LIN {X -90.429,Y -7.308,Z -76.160,A -90.000,B 90.000,C 0.000} C_DIS
LIN {X -90.430,Y -7.308,Z -76.160,A -90.000,B 90.000,C 0.000} C_DIS
LIN {X -90.438,Y -7.308,Z -76.159,A -90.000,B 90.000,C 0.000} C_DIS
LIN {X -90.556,Y -7.308,Z -76.141,A -90.000,B 90.000,C 0.000} C_DIS
LIN {X -90.743,Y -7.308,Z -76.119,A -90.000,B 90.000,C 0.000} C_DIS
LIN {X -90.835,Y -7.308,Z -76.112,A -90.000,B 90.000,C 0.000} C_DIS
LIN {X -90.996,Y -7.308,Z -76.109,A -90.000,B 90.000,C 0.000} C_DIS
LIN {X -91.021,Y -7.308,Z -76.109,A -90.000,B 90.000,C 0.000} C_DIS
LIN {X -91.083,Y -7.308,Z -76.111,A -90.000,B 90.000,C 0.000} C_DIS
LIN {X -91.127,Y -7.308,Z -76.111,A -90.000,B 90.000,C 0.000} C_DIS
LIN {X -91.716,Y -7.308,Z -76.119,A -90.000,B 90.000,C 0.000} C_DIS
LIN {X -91.719,Y -7.308,Z -76.119,A -90.000,B 90.000,C 0.000} C_DIS
LIN {X -91.850,Y -7.308,Z -76.127,A -90.000,B 90.000,C 0.000} C_DIS
LIN {X -91.854,Y -7.308,Z -76.127,A -90.000,B 90.000,C 0.000} C_DIS
LIN {X -91.855,Y -7.308,Z -76.127,A -90.000,B 90.000,C 0.000} C_DIS
LIN {X -92.275,Y -7.308,Z -76.134,A -90.000,B 90.000,C 0.000} C_DIS
LIN {X -92.401,Y -7.308,Z -76.144,A -90.000,B 90.000,C 0.000} C_DIS
LIN {X -92.567,Y -7.308,Z -76.154,A -90.000,B 90.000,C 0.000} C_DIS
LIN {X -92.855,Y -7.308,Z -76.172,A -90.000,B 90.000,C 0.000} C_DIS
LIN {X -93.155,Y -7.308,Z -76.171,A -90.000,B 90.000,C 0.000} C_DIS
LIN {X -93.950,Y -7.308,Z -76.211,A -90.000,B 90.000,C 0.000} C_DIS
LIN {X -93.975,Y -7.308,Z -76.209,A -90.000,B 90.000,C 0.000} C_DIS
LIN {X -94.009,Y -7.308,Z -76.208,A -90.000,B 90.000,C 0.000} C_DIS
LIN {X -94.203,Y -7.308,Z -76.206,A -90.000,B 90.000,C 0.000} C_DIS
LIN {X -94.938,Y -7.308,Z -76.181,A -90.000,B 90.000,C 0.000} C_DIS
LIN {X -95.138,Y -7.308,Z -76.181,A -90.000,B 90.000,C 0.000} C_DIS
LIN {X -95.500,Y -7.308,Z -76.164,A -90.000,B 90.000,C 0.000} C_DIS
LIN {X -95.593,Y -7.308,Z -76.159,A -90.000,B 90.000,C 0.000} C_DIS
LIN {X -96.438,Y -7.308,Z -76.050,A -90.000,B 90.000,C 0.000} C_DIS
LIN {X -96.876,Y -7.308,Z -76.007,A -90.000,B 90.000,C 0.000} C_DIS
LIN {X -97.150,Y -7.308,Z -75.964,A -90.000,B 90.000,C 0.000} C_DIS
LIN {X -97.326,Y -7.308,Z -75.936,A -90.000,B 90.000,C 0.000} C_DIS
LIN {X -98.066,Y -7.308,Z -75.745,A -90.000,B 90.000,C 0.000} C_DIS
LIN {X -98.704,Y -7.308,Z -75.598,A -90.000,B 90.000,C 0.000} C_DIS
LIN {X -98.924,Y -7.308,Z -75.538,A -90.000,B 90.000,C 0.000} C_DIS
LIN {X -99.143,Y -7.308,Z -75.478,A -90.000,B 90.000,C 0.000} C_DIS
LIN {X -99.355,Y -7.308,Z -75.394,A -90.000,B 90.000,C 0.000} C_DIS
LIN {X -99.566,Y -7.308,Z -75.311,A -90.000,B 90.000,C 0.000} C_DIS
LIN {X -100.148,Y -7.308,Z -75.070,A -90.000,B 90.000,C 0.000} C_DIS
LIN {X -100.612,Y -7.308,Z -74.890,A -90.000,B 90.000,C 0.000} C_DIS
LIN {X -100.815,Y -7.308,Z -74.810,A -90.000,B 90.000,C 0.000} C_DIS
LIN {X -101.035,Y -7.308,Z -74.723,A -90.000,B 90.000,C 0.000} C_DIS
LIN {X -101.228,Y -7.308,Z -74.620,A -90.000,B 90.000,C 0.000} C_DIS
LIN {X -101.438,Y -7.308,Z -74.510,A -90.000,B 90.000,C 0.000} C_DIS
LIN {X -102.233,Y -7.308,Z -74.035,A -90.000,B 90.000,C 0.000} C_DIS
LIN {X -102.984,Y -7.308,Z -73.608,A -90.000,B 90.000,C 0.000} C_DIS
LIN {X -103.195,Y -7.308,Z -73.465,A -90.000,B 90.000,C 0.000} C_DIS
LIN {X -103.361,Y -7.308,Z -73.353,A -90.000,B 90.000,C 0.000} C_DIS
LIN {X -104.367,Y -7.308,Z -72.602,A -90.000,B 90.000,C 0.000} C_DIS
LIN {X -104.886,Y -7.308,Z -72.231,A -90.000,B 90.000,C 0.000} C_DIS
LIN {X -105.135,Y -7.308,Z -72.019,A -90.000,B 90.000,C 0.000} C_DIS
LIN {X -105.233,Y -7.308,Z -71.935,A -90.000,B 90.000,C 0.000} C_DIS
LIN {X -106.016,Y -7.308,Z -71.241,A -90.000,B 90.000,C 0.000} C_DIS
LIN {X -106.511,Y -7.308,Z -70.803,A -90.000,B 90.000,C 0.000} C_DIS
LIN {X -106.623,Y -7.308,Z -70.708,A -90.000,B 90.000,C 0.000} C_DIS
LIN {X -106.647,Y -7.308,Z -70.687,A -90.000,B 90.000,C 0.000} C_DIS
LIN {X -107.011,Y -7.308,Z -70.310,A -90.000,B 90.000,C 0.000} C_DIS
LIN {X -107.247,Y -7.308,Z -70.060,A -90.000,B 90.000,C 0.000} C_DIS
LIN {X -107.570,Y -7.308,Z -69.717,A -90.000,B 90.000,C 0.000} C_DIS
LIN {X -107.658,Y -7.308,Z -69.623,A -90.000,B 90.000,C 0.000} C_DIS
LIN {X -107.961,Y -7.308,Z -69.302,A -90.000,B 90.000,C 0.000} C_DIS
LIN {X -108.119,Y -7.308,Z -69.134,A -90.000,B 90.000,C 0.000} C_DIS
LIN {X -108.189,Y -7.308,Z -69.054,A -90.000,B 90.000,C 0.000} C_DIS
LIN {X -108.324,Y -7.308,Z -68.876,A -90.000,B 90.000,C 0.000} C_DIS
LIN {X -108.394,Y -7.308,Z -68.788,A -90.000,B 90.000,C 0.000} C_DIS
LIN {X -108.549,Y -7.308,Z -68.594,A -90.000,B 90.000,C 0.000} C_DIS
LIN {X -108.807,Y -7.308,Z -68.269,A -90.000,B 90.000,C 0.000} C_DIS
LIN {X -109.048,Y -7.308,Z -67.965,A -90.000,B 90.000,C 0.000} C_DIS
LIN {X -109.050,Y -7.308,Z -67.962,A -90.000,B 90.000,C 0.000} C_DIS
LIN {X -109.051,Y -7.308,Z -67.961,A -90.000,B 90.000,C 0.000} C_DIS
LIN {X -109.057,Y -7.308,Z -67.953,A -90.000,B 90.000,C 0.000} C_DIS
LIN {X -109.064,Y -7.308,Z -67.944,A -90.000,B 90.000,C 0.000} C_DIS
LIN {X -109.315,Y -7.308,Z -67.619,A -90.000,B 90.000,C 0.000} C_DIS
LIN {X -109.317,Y -7.308,Z -67.616,A -90.000,B 90.000,C 0.000} C_DIS
LIN {X -109.330,Y -7.308,Z -67.598,A -90.000,B 90.000,C 0.000} C_DIS
LIN {X -109.445,Y -7.308,Z -67.437,A -90.000,B 90.000,C 0.000} C_DIS
LIN {X -109.557,Y -7.308,Z -67.257,A -90.000,B 90.000,C 0.000} C_DIS
LIN {X -109.624,Y -7.308,Z -67.149,A -90.000,B 90.000,C 0.000} C_DIS
LIN {X -109.859,Y -7.308,Z -66.772,A -90.000,B 90.000,C 0.000} C_DIS
LIN {X -110.128,Y -7.308,Z -66.355,A -90.000,B 90.000,C 0.000} C_DIS
LIN {X -110.187,Y -7.308,Z -66.262,A -90.000,B 90.000,C 0.000} C_DIS
LIN {X -110.241,Y -7.308,Z -66.176,A -90.000,B 90.000,C 0.000} C_DIS
LIN {X -110.406,Y -7.308,Z -65.897,A -90.000,B 90.000,C 0.000} C_DIS
LIN {X -110.474,Y -7.308,Z -65.784,A -90.000,B 90.000,C 0.000} C_DIS
LIN {X -111.122,Y -7.308,Z -64.499,A -90.000,B 90.000,C 0.000} C_DIS
LIN {X -111.141,Y -7.308,Z -64.462,A -90.000,B 90.000,C 0.000} C_DIS
LIN {X -111.142,Y -7.308,Z -64.459,A -90.000,B 90.000,C 0.000} C_DIS
LIN {X -111.143,Y -7.308,Z -64.457,A -90.000,B 90.000,C 0.000} C_DIS
LIN {X -111.144,Y -7.308,Z -64.456,A -90.000,B 90.000,C 0.000} C_DIS
LIN {X -111.144,Y -7.308,Z -64.455,A -90.000,B 90.000,C 0.000} C_DIS
LIN {X -111.330,Y -7.308,Z -64.046,A -90.000,B 90.000,C 0.000} C_DIS
LIN {X -111.330,Y -7.308,Z -64.044,A -90.000,B 90.000,C 0.000} C_DIS
LIN {X -111.331,Y -7.308,Z -64.041,A -90.000,B 90.000,C 0.000} C_DIS
LIN {X -111.339,Y -7.308,Z -64.023,A -90.000,B 90.000,C 0.000} C_DIS
LIN {X -111.858,Y -7.308,Z -62.803,A -90.000,B 90.000,C 0.000} C_DIS
LIN {X -111.946,Y -7.308,Z -62.595,A -90.000,B 90.000,C 0.000} C_DIS
LIN {X -111.980,Y -7.308,Z -62.501,A -90.000,B 90.000,C 0.000} C_DIS
LIN {X -112.247,Y -7.308,Z -61.757,A -90.000,B 90.000,C 0.000} C_DIS
LIN {X -112.297,Y -7.308,Z -61.622,A -90.000,B 90.000,C 0.000} C_DIS
LIN {X -112.357,Y -7.308,Z -61.457,A -90.000,B 90.000,C 0.000} C_DIS
LIN {X -112.381,Y -7.308,Z -61.394,A -90.000,B 90.000,C 0.000} C_DIS
LIN {X -112.489,Y -7.308,Z -61.121,A -90.000,B 90.000,C 0.000} C_DIS
LIN {X -112.498,Y -7.308,Z -61.099,A -90.000,B 90.000,C 0.000} C_DIS
LIN {X -112.511,Y -7.308,Z -61.065,A -90.000,B 90.000,C 0.000} C_DIS
LIN {X -112.548,Y -7.308,Z -60.970,A -90.000,B 90.000,C 0.000} C_DIS
LIN {X -112.569,Y -7.308,Z -60.913,A -90.000,B 90.000,C 0.000} C_DIS
LIN {X -112.574,Y -7.308,Z -60.900,A -90.000,B 90.000,C 0.000} C_DIS
LIN {X -112.579,Y -7.308,Z -60.889,A -90.000,B 90.000,C 0.000} C_DIS
LIN {X -112.589,Y -7.308,Z -60.860,A -90.000,B 90.000,C 0.000} C_DIS
LIN {X -112.641,Y -7.308,Z -60.721,A -90.000,B 90.000,C 0.000} C_DIS
LIN {X -112.737,Y -7.308,Z -60.464,A -90.000,B 90.000,C 0.000} C_DIS
LIN {X -112.752,Y -7.308,Z -60.423,A -90.000,B 90.000,C 0.000} C_DIS
LIN {X -112.766,Y -7.308,Z -60.386,A -90.000,B 90.000,C 0.000} C_DIS
LIN {X -112.917,Y -7.308,Z -59.968,A -90.000,B 90.000,C 0.000} C_DIS
LIN {X -112.929,Y -7.308,Z -59.935,A -90.000,B 90.000,C 0.000} C_DIS
LIN {X -112.957,Y -7.308,Z -59.850,A -90.000,B 90.000,C 0.000} C_DIS
LIN {X -113.226,Y -7.308,Z -59.066,A -90.000,B 90.000,C 0.000} C_DIS
LIN {X -113.275,Y -7.308,Z -58.928,A -90.000,B 90.000,C 0.000} C_DIS
LIN {X -113.292,Y -7.308,Z -58.880,A -90.000,B 90.000,C 0.000} C_DIS
LIN {X -113.430,Y -7.308,Z -58.480,A -90.000,B 90.000,C 0.000} C_DIS
LIN {X -113.480,Y -7.308,Z -58.334,A -90.000,B 90.000,C 0.000} C_DIS
LIN {X -113.651,Y -7.308,Z -57.841,A -90.000,B 90.000,C 0.000} C_DIS
LIN {X -113.725,Y -7.308,Z -57.605,A -90.000,B 90.000,C 0.000} C_DIS
LIN {X -113.775,Y -7.308,Z -57.446,A -90.000,B 90.000,C 0.000} C_DIS
LIN {X -113.840,Y -7.308,Z -57.265,A -90.000,B 90.000,C 0.000} C_DIS
LIN {X -113.863,Y -7.308,Z -57.201,A -90.000,B 90.000,C 0.000} C_DIS
LIN {X -113.998,Y -7.308,Z -56.823,A -90.000,B 90.000,C 0.000} C_DIS
LIN {X -114.035,Y -7.308,Z -56.712,A -90.000,B 90.000,C 0.000} C_DIS
LIN {X -114.077,Y -7.308,Z -56.590,A -90.000,B 90.000,C 0.000} C_DIS
LIN {X -114.087,Y -7.308,Z -56.561,A -90.000,B 90.000,C 0.000} C_DIS
LIN {X -114.176,Y -7.308,Z -56.299,A -90.000,B 90.000,C 0.000} C_DIS
LIN {X -114.177,Y -7.308,Z -56.295,A -90.000,B 90.000,C 0.000} C_DIS
LIN {X -114.260,Y -7.308,Z -56.079,A -90.000,B 90.000,C 0.000} C_DIS
LIN {X -114.595,Y -7.308,Z -55.238,A -90.000,B 90.000,C 0.000} C_DIS
LIN {X -114.855,Y -7.308,Z -54.587,A -90.000,B 90.000,C 0.000} C_DIS
LIN {X -115.040,Y -7.308,Z -54.138,A -90.000,B 90.000,C 0.000} C_DIS
LIN {X -115.335,Y -7.308,Z -53.342,A -90.000,B 90.000,C 0.000} C_DIS
LIN {X -115.406,Y -7.308,Z -53.154,A -90.000,B 90.000,C 0.000} C_DIS
LIN {X -115.537,Y -7.308,Z -52.781,A -90.000,B 90.000,C 0.000} C_DIS
LIN {X -115.545,Y -7.308,Z -52.758,A -90.000,B 90.000,C 0.000} C_DIS
LIN {X -115.549,Y -7.308,Z -52.745,A -90.000,B 90.000,C 0.000} C_DIS
LIN {X -115.560,Y -7.308,Z -52.713,A -90.000,B 90.000,C 0.000} C_DIS
LIN {X -115.573,Y -7.308,Z -52.666,A -90.000,B 90.000,C 0.000} C_DIS
LIN {X -115.577,Y -7.308,Z -52.655,A -90.000,B 90.000,C 0.000} C_DIS
LIN {X -115.783,Y -7.308,Z -51.915,A -90.000,B 90.000,C 0.000} C_DIS
LIN {X -115.800,Y -7.308,Z -51.855,A -90.000,B 90.000,C 0.000} C_DIS
LIN {X -115.805,Y -7.308,Z -51.837,A -90.000,B 90.000,C 0.000} C_DIS
LIN {X -115.851,Y -7.308,Z -51.672,A -90.000,B 90.000,C 0.000} C_DIS
LIN {X -115.877,Y -7.308,Z -51.578,A -90.000,B 90.000,C 0.000} C_DIS
LIN {X -115.919,Y -7.308,Z -51.379,A -90.000,B 90.000,C 0.000} C_DIS
LIN {X -115.971,Y -7.308,Z -51.132,A -90.000,B 90.000,C 0.000} C_DIS
LIN {X -115.990,Y -7.308,Z -50.930,A -90.000,B 90.000,C 0.000} C_DIS
LIN {X -115.995,Y -7.308,Z -50.884,A -90.000,B 90.000,C 0.000} C_DIS
LIN {X -116.015,Y -7.308,Z -50.679,A -90.000,B 90.000,C 0.000} C_DIS
LIN {X -116.038,Y -7.308,Z -50.413,A -90.000,B 90.000,C 0.000} C_DIS
LIN {X -116.044,Y -7.308,Z -50.351,A -90.000,B 90.000,C 0.000} C_DIS
LIN {X -116.053,Y -7.308,Z -50.262,A -90.000,B 90.000,C 0.000} C_DIS
LIN {X -116.072,Y -7.308,Z -50.070,A -90.000,B 90.000,C 0.000} C_DIS
LIN {X -116.088,Y -7.308,Z -49.898,A -90.000,B 90.000,C 0.000} C_DIS
LIN {X -116.085,Y -7.308,Z -49.616,A -90.000,B 90.000,C 0.000} C_DIS
LIN {X -116.082,Y -7.308,Z -49.442,A -90.000,B 90.000,C 0.000} C_DIS
LIN {X -116.079,Y -7.308,Z -49.392,A -90.000,B 90.000,C 0.000} C_DIS
LIN {X -116.077,Y -7.308,Z -49.365,A -90.000,B 90.000,C 0.000} C_DIS
LIN {X -116.068,Y -7.308,Z -49.205,A -90.000,B 90.000,C 0.000} C_DIS
LIN {X -116.055,Y -7.308,Z -48.764,A -90.000,B 90.000,C 0.000} C_DIS
LIN {X -116.049,Y -7.308,Z -48.715,A -90.000,B 90.000,C 0.000} C_DIS
LIN {X -116.049,Y -7.308,Z -48.713,A -90.000,B 90.000,C 0.000} C_DIS
LIN {X -116.045,Y -7.308,Z -48.687,A -90.000,B 90.000,C 0.000} C_DIS
LIN {X -116.046,Y -7.308,Z -48.684,A -90.000,B 90.000,C 0.000} C_DIS
LIN {X -116.102,Y -7.308,Z -48.546,A -90.000,B 90.000,C 0.000} C_DIS
LIN {X -116.109,Y -7.308,Z -48.529,A -90.000,B 90.000,C 0.000} C_DIS
LIN {X -116.231,Y -7.308,Z -48.216,A -90.000,B 90.000,C 0.000} C_DIS
LIN {X -116.273,Y -7.308,Z -48.106,A -90.000,B 90.000,C 0.000} C_DIS
LIN {X -116.402,Y -7.308,Z -47.760,A -90.000,B 90.000,C 0.000} C_DIS
LIN {X -116.428,Y -7.308,Z -47.687,A -90.000,B 90.000,C 0.000} C_DIS
LIN {X -116.462,Y -7.308,Z -47.594,A -90.000,B 90.000,C 0.000} C_DIS
LIN {X -116.577,Y -7.308,Z -47.256,A -90.000,B 90.000,C 0.000} C_DIS
LIN {X -116.682,Y -7.308,Z -46.928,A -90.000,B 90.000,C 0.000} C_DIS
LIN {X -116.712,Y -7.308,Z -46.836,A -90.000,B 90.000,C 0.000} C_DIS
LIN {X -116.738,Y -7.308,Z -46.742,A -90.000,B 90.000,C 0.000} C_DIS
LIN {X -116.816,Y -7.308,Z -46.454,A -90.000,B 90.000,C 0.000} C_DIS
LIN {X -116.874,Y -7.308,Z -46.240,A -90.000,B 90.000,C 0.000} C_DIS
LIN {X -116.912,Y -7.308,Z -46.079,A -90.000,B 90.000,C 0.000} C_DIS
LIN {X -116.977,Y -7.308,Z -45.819,A -90.000,B 90.000,C 0.000} C_DIS
LIN {X -117.000,Y -7.308,Z -45.688,A -90.000,B 90.000,C 0.000} C_DIS
LIN {X -117.032,Y -7.308,Z -45.502,A -90.000,B 90.000,C 0.000} C_DIS
LIN {X -117.066,Y -7.308,Z -45.295,A -90.000,B 90.000,C 0.000} C_DIS
LIN {X -117.091,Y -7.308,Z -45.116,A -90.000,B 90.000,C 0.000} C_DIS
LIN {X -117.122,Y -7.308,Z -44.884,A -90.000,B 90.000,C 0.000} C_DIS
LIN {X -117.154,Y -7.308,Z -44.619,A -90.000,B 90.000,C 0.000} C_DIS
LIN {X -117.172,Y -7.308,Z -44.476,A -90.000,B 90.000,C 0.000} C_DIS
LIN {X -117.184,Y -7.308,Z -44.378,A -90.000,B 90.000,C 0.000} C_DIS
LIN {X -117.189,Y -7.308,Z -44.049,A -90.000,B 90.000,C 0.000} C_DIS
LIN {X -117.191,Y -7.308,Z -43.922,A -90.000,B 90.000,C 0.000} C_DIS
LIN {X -117.191,Y -7.308,Z -43.911,A -90.000,B 90.000,C 0.000} C_DIS
LIN {X -117.188,Y -7.308,Z -43.790,A -90.000,B 90.000,C 0.000} C_DIS
LIN {X -117.187,Y -7.308,Z -43.750,A -90.000,B 90.000,C 0.000} C_DIS
LIN {X -117.190,Y -7.308,Z -43.518,A -90.000,B 90.000,C 0.000} C_DIS
LIN {X -117.191,Y -7.308,Z -43.491,A -90.000,B 90.000,C 0.000} C_DIS
LIN {X -117.191,Y -7.308,Z -43.489,A -90.000,B 90.000,C 0.000} C_DIS
LIN {X -117.190,Y -7.308,Z -43.459,A -90.000,B 90.000,C 0.000} C_DIS
LIN {X -117.185,Y -7.308,Z -43.036,A -90.000,B 90.000,C 0.000} C_DIS
LIN {X -117.181,Y -7.308,Z -43.004,A -90.000,B 90.000,C 0.000} C_DIS
LIN {X -117.153,Y -7.308,Z -42.780,A -90.000,B 90.000,C 0.000} C_DIS
LIN {X -117.137,Y -7.308,Z -42.642,A -90.000,B 90.000,C 0.000} C_DIS
LIN {X -117.132,Y -7.308,Z -42.602,A -90.000,B 90.000,C 0.000} C_DIS
LIN {X -117.129,Y -7.308,Z -42.575,A -90.000,B 90.000,C 0.000} C_DIS
LIN {X -117.082,Y -7.308,Z -42.199,A -90.000,B 90.000,C 0.000} C_DIS
LIN {X -117.072,Y -7.308,Z -42.126,A -90.000,B 90.000,C 0.000} C_DIS
LIN {X -117.040,Y -7.308,Z -41.945,A -90.000,B 90.000,C 0.000} C_DIS
LIN {X -117.020,Y -7.308,Z -41.836,A -90.000,B 90.000,C 0.000} C_DIS
LIN {X -116.975,Y -7.308,Z -41.649,A -90.000,B 90.000,C 0.000} C_DIS
LIN {X -116.937,Y -7.308,Z -41.456,A -90.000,B 90.000,C 0.000} C_DIS
LIN {X -116.879,Y -7.308,Z -41.233,A -90.000,B 90.000,C 0.000} C_DIS
LIN {X -116.827,Y -7.308,Z -41.029,A -90.000,B 90.000,C 0.000} C_DIS
LIN {X -116.765,Y -7.308,Z -40.854,A -90.000,B 90.000,C 0.000} C_DIS
LIN {X -116.712,Y -7.308,Z -40.691,A -90.000,B 90.000,C 0.000} C_DIS
LIN {X -116.681,Y -7.308,Z -40.605,A -90.000,B 90.000,C 0.000} C_DIS
LIN {X -116.625,Y -7.308,Z -40.452,A -90.000,B 90.000,C 0.000} C_DIS
LIN {X -116.619,Y -7.308,Z -40.436,A -90.000,B 90.000,C 0.000} C_DIS
LIN {X -116.522,Y -7.308,Z -40.182,A -90.000,B 90.000,C 0.000} C_DIS
LIN {X -116.520,Y -7.308,Z -40.178,A -90.000,B 90.000,C 0.000} C_DIS
LIN {X -116.529,Y -7.308,Z -40.156,A -90.000,B 90.000,C 0.000} C_DIS
LIN {X -116.555,Y -7.308,Z -40.093,A -90.000,B 90.000,C 0.000} C_DIS
LIN {X -116.680,Y -7.308,Z -39.786,A -90.000,B 90.000,C 0.000} C_DIS
LIN {X -116.713,Y -7.308,Z -39.703,A -90.000,B 90.000,C 0.000} C_DIS
LIN {X -116.734,Y -7.308,Z -39.651,A -90.000,B 90.000,C 0.000} C_DIS
LIN {X -116.788,Y -7.308,Z -39.504,A -90.000,B 90.000,C 0.000} C_DIS
LIN {X -116.887,Y -7.308,Z -39.234,A -90.000,B 90.000,C 0.000} C_DIS
LIN {X -116.969,Y -7.308,Z -38.990,A -90.000,B 90.000,C 0.000} C_DIS
LIN {X -117.042,Y -7.308,Z -38.777,A -90.000,B 90.000,C 0.000} C_DIS
LIN {X -117.100,Y -7.308,Z -38.586,A -90.000,B 90.000,C 0.000} C_DIS
LIN {X -117.151,Y -7.308,Z -38.421,A -90.000,B 90.000,C 0.000} C_DIS
LIN {X -117.191,Y -7.308,Z -38.265,A -90.000,B 90.000,C 0.000} C_DIS
LIN {X -117.259,Y -7.308,Z -37.996,A -90.000,B 90.000,C 0.000} C_DIS
LIN {X -117.295,Y -7.308,Z -37.837,A -90.000,B 90.000,C 0.000} C_DIS
LIN {X -117.321,Y -7.308,Z -37.718,A -90.000,B 90.000,C 0.000} C_DIS
LIN {X -117.354,Y -7.308,Z -37.563,A -90.000,B 90.000,C 0.000} C_DIS
LIN {X -117.363,Y -7.308,Z -37.510,A -90.000,B 90.000,C 0.000} C_DIS
LIN {X -117.368,Y -7.308,Z -37.480,A -90.000,B 90.000,C 0.000} C_DIS
LIN {X -117.422,Y -7.308,Z -37.158,A -90.000,B 90.000,C 0.000} C_DIS
LIN {X -117.446,Y -7.308,Z -37.010,A -90.000,B 90.000,C 0.000} C_DIS
LIN {X -117.458,Y -7.308,Z -36.909,A -90.000,B 90.000,C 0.000} C_DIS
LIN {X -117.482,Y -7.308,Z -36.721,A -90.000,B 90.000,C 0.000} C_DIS
LIN {X -117.498,Y -7.308,Z -36.449,A -90.000,B 90.000,C 0.000} C_DIS
LIN {X -117.511,Y -7.308,Z -36.246,A -90.000,B 90.000,C 0.000} C_DIS
LIN {X -117.516,Y -7.308,Z -36.108,A -90.000,B 90.000,C 0.000} C_DIS
LIN {X -117.526,Y -7.308,Z -35.954,A -90.000,B 90.000,C 0.000} C_DIS
LIN {X -117.526,Y -7.308,Z -35.796,A -90.000,B 90.000,C 0.000} C_DIS
LIN {X -117.526,Y -7.308,Z -35.502,A -90.000,B 90.000,C 0.000} C_DIS
LIN {X -117.525,Y -7.308,Z -35.472,A -90.000,B 90.000,C 0.000} C_DIS
LIN {X -117.519,Y -7.308,Z -35.299,A -90.000,B 90.000,C 0.000} C_DIS
LIN {X -117.512,Y -7.308,Z -35.158,A -90.000,B 90.000,C 0.000} C_DIS
LIN {X -117.482,Y -7.308,Z -34.830,A -90.000,B 90.000,C 0.000} C_DIS
LIN {X -117.472,Y -7.308,Z -34.736,A -90.000,B 90.000,C 0.000} C_DIS
LIN {X -117.467,Y -7.308,Z -34.687,A -90.000,B 90.000,C 0.000} C_DIS
LIN {X -117.463,Y -7.308,Z -34.659,A -90.000,B 90.000,C 0.000} C_DIS
LIN {X -117.459,Y -7.308,Z -34.620,A -90.000,B 90.000,C 0.000} C_DIS
LIN {X -117.442,Y -7.308,Z -34.475,A -90.000,B 90.000,C 0.000} C_DIS
LIN {X -117.433,Y -7.308,Z -34.401,A -90.000,B 90.000,C 0.000} C_DIS
LIN {X -117.419,Y -7.308,Z -34.331,A -90.000,B 90.000,C 0.000} C_DIS
LIN {X -117.381,Y -7.308,Z -34.119,A -90.000,B 90.000,C 0.000} C_DIS
LIN {X -117.317,Y -7.308,Z -33.800,A -90.000,B 90.000,C 0.000} C_DIS
LIN {X -117.289,Y -7.308,Z -33.661,A -90.000,B 90.000,C 0.000} C_DIS
LIN {X -117.244,Y -7.308,Z -33.481,A -90.000,B 90.000,C 0.000} C_DIS
LIN {X -117.218,Y -7.308,Z -33.387,A -90.000,B 90.000,C 0.000} C_DIS
LIN {X -117.167,Y -7.308,Z -33.226,A -90.000,B 90.000,C 0.000} C_DIS
LIN {X -117.083,Y -7.308,Z -32.959,A -90.000,B 90.000,C 0.000} C_DIS
LIN {X -117.026,Y -7.308,Z -32.780,A -90.000,B 90.000,C 0.000} C_DIS
LIN {X -116.990,Y -7.308,Z -32.673,A -90.000,B 90.000,C 0.000} C_DIS
LIN {X -116.936,Y -7.308,Z -32.528,A -90.000,B 90.000,C 0.000} C_DIS
LIN {X -116.902,Y -7.308,Z -32.443,A -90.000,B 90.000,C 0.000} C_DIS
LIN {X -116.846,Y -7.308,Z -32.302,A -90.000,B 90.000,C 0.000} C_DIS
LIN {X -116.751,Y -7.308,Z -32.064,A -90.000,B 90.000,C 0.000} C_DIS
LIN {X -116.746,Y -7.308,Z -32.052,A -90.000,B 90.000,C 0.000} C_DIS
LIN {X -116.634,Y -7.308,Z -31.804,A -90.000,B 90.000,C 0.000} C_DIS
LIN {X -116.634,Y -7.308,Z -31.803,A -90.000,B 90.000,C 0.000} C_DIS
LIN {X -116.633,Y -7.308,Z -31.801,A -90.000,B 90.000,C 0.000} C_DIS
LIN {X -116.436,Y -7.308,Z -31.397,A -90.000,B 90.000,C 0.000} C_DIS
LIN {X -116.436,Y -7.308,Z -31.395,A -90.000,B 90.000,C 0.000} C_DIS
LIN {X -116.435,Y -7.308,Z -31.395,A -90.000,B 90.000,C 0.000} C_DIS
LIN {X -116.422,Y -7.308,Z -31.367,A -90.000,B 90.000,C 0.000} C_DIS
LIN {X -116.320,Y -7.308,Z -31.161,A -90.000,B 90.000,C 0.000} C_DIS
LIN {X -116.309,Y -7.308,Z -31.142,A -90.000,B 90.000,C 0.000} C_DIS
LIN {X -116.188,Y -7.308,Z -30.931,A -90.000,B 90.000,C 0.000} C_DIS
LIN {X -116.153,Y -7.308,Z -30.870,A -90.000,B 90.000,C 0.000} C_DIS
LIN {X -115.947,Y -7.308,Z -30.543,A -90.000,B 90.000,C 0.000} C_DIS
LIN {X -115.922,Y -7.308,Z -30.506,A -90.000,B 90.000,C 0.000} C_DIS
LIN {X -115.794,Y -7.308,Z -30.316,A -90.000,B 90.000,C 0.000} C_DIS
LIN {X -115.776,Y -7.308,Z -30.289,A -90.000,B 90.000,C 0.000} C_DIS
LIN {X -115.768,Y -7.308,Z -30.277,A -90.000,B 90.000,C 0.000} C_DIS
LIN {X -115.751,Y -7.308,Z -30.253,A -90.000,B 90.000,C 0.000} C_DIS
LIN {X -115.496,Y -7.308,Z -29.933,A -90.000,B 90.000,C 0.000} C_DIS
LIN {X -115.468,Y -7.308,Z -29.897,A -90.000,B 90.000,C 0.000} C_DIS
LIN {X -115.297,Y -7.308,Z -29.688,A -90.000,B 90.000,C 0.000} C_DIS
LIN {X -115.272,Y -7.308,Z -29.657,A -90.000,B 90.000,C 0.000} C_DIS
LIN {X -114.993,Y -7.308,Z -29.376,A -90.000,B 90.000,C 0.000} C_DIS
LIN {X -114.951,Y -7.308,Z -29.334,A -90.000,B 90.000,C 0.000} C_DIS
LIN {X -114.920,Y -7.308,Z -29.303,A -90.000,B 90.000,C 0.000} C_DIS
LIN {X -114.722,Y -7.308,Z -29.105,A -90.000,B 90.000,C 0.000} C_DIS
LIN {X -114.681,Y -7.308,Z -29.066,A -90.000,B 90.000,C 0.000} C_DIS
LIN {X -114.489,Y -7.308,Z -28.886,A -90.000,B 90.000,C 0.000} C_DIS
LIN {X -114.460,Y -7.308,Z -28.852,A -90.000,B 90.000,C 0.000} C_DIS
LIN {X -114.446,Y -7.308,Z -28.835,A -90.000,B 90.000,C 0.000} C_DIS
LIN {X -114.406,Y -7.308,Z -28.790,A -90.000,B 90.000,C 0.000} C_DIS
LIN {X -114.340,Y -7.308,Z -28.697,A -90.000,B 90.000,C 0.000} C_DIS
LIN {X -114.321,Y -7.308,Z -28.671,A -90.000,B 90.000,C 0.000} C_DIS
LIN {X -114.300,Y -7.308,Z -28.640,A -90.000,B 90.000,C 0.000} C_DIS
LIN {X -114.205,Y -7.308,Z -28.492,A -90.000,B 90.000,C 0.000} C_DIS
LIN {X -114.104,Y -7.308,Z -28.333,A -90.000,B 90.000,C 0.000} C_DIS
LIN {X -114.004,Y -7.308,Z -28.175,A -90.000,B 90.000,C 0.000} C_DIS
LIN {X -113.925,Y -7.308,Z -28.049,A -90.000,B 90.000,C 0.000} C_DIS
LIN {X -113.897,Y -7.308,Z -28.005,A -90.000,B 90.000,C 0.000} C_DIS
LIN {X -113.813,Y -7.308,Z -27.871,A -90.000,B 90.000,C 0.000} C_DIS
LIN {X -113.727,Y -7.308,Z -27.736,A -90.000,B 90.000,C 0.000} C_DIS
LIN {X -113.688,Y -7.308,Z -27.674,A -90.000,B 90.000,C 0.000} C_DIS
LIN {X -113.475,Y -7.308,Z -27.351,A -90.000,B 90.000,C 0.000} C_DIS
LIN {X -113.379,Y -7.308,Z -27.199,A -90.000,B 90.000,C 0.000} C_DIS
LIN {X -113.154,Y -7.308,Z -26.894,A -90.000,B 90.000,C 0.000} C_DIS
LIN {X -113.043,Y -7.308,Z -26.735,A -90.000,B 90.000,C 0.000} C_DIS
LIN {X -112.857,Y -7.308,Z -26.502,A -90.000,B 90.000,C 0.000} C_DIS
LIN {X -112.759,Y -7.308,Z -26.379,A -90.000,B 90.000,C 0.000} C_DIS
LIN {X -112.719,Y -7.308,Z -26.330,A -90.000,B 90.000,C 0.000} C_DIS
LIN {X -112.547,Y -7.308,Z -26.121,A -90.000,B 90.000,C 0.000} C_DIS
LIN {X -112.499,Y -7.308,Z -26.061,A -90.000,B 90.000,C 0.000} C_DIS
LIN {X -112.395,Y -7.308,Z -25.931,A -90.000,B 90.000,C 0.000} C_DIS
LIN {X -112.146,Y -7.308,Z -25.663,A -90.000,B 90.000,C 0.000} C_DIS
LIN {X -112.003,Y -7.308,Z -25.505,A -90.000,B 90.000,C 0.000} C_DIS
LIN {X -111.924,Y -7.308,Z -25.421,A -90.000,B 90.000,C 0.000} C_DIS
LIN {X -111.820,Y -7.308,Z -25.311,A -90.000,B 90.000,C 0.000} C_DIS
LIN {X -111.741,Y -7.308,Z -25.237,A -90.000,B 90.000,C 0.000} C_DIS
LIN {X -111.401,Y -7.308,Z -24.914,A -90.000,B 90.000,C 0.000} C_DIS
LIN {X -111.341,Y -7.308,Z -24.857,A -90.000,B 90.000,C 0.000} C_DIS
LIN {X -111.080,Y -7.308,Z -24.612,A -90.000,B 90.000,C 0.000} C_DIS
LIN {X -110.993,Y -7.308,Z -24.541,A -90.000,B 90.000,C 0.000} C_DIS
LIN {X -110.629,Y -7.308,Z -24.251,A -90.000,B 90.000,C 0.000} C_DIS
LIN {X -110.555,Y -7.308,Z -24.196,A -90.000,B 90.000,C 0.000} C_DIS
LIN {X -110.275,Y -7.308,Z -23.988,A -90.000,B 90.000,C 0.000} C_DIS
LIN {X -110.166,Y -7.308,Z -23.914,A -90.000,B 90.000,C 0.000} C_DIS
LIN {X -109.779,Y -7.308,Z -23.661,A -90.000,B 90.000,C 0.000} C_DIS
LIN {X -109.684,Y -7.308,Z -23.605,A -90.000,B 90.000,C 0.000} C_DIS
LIN {X -109.398,Y -7.308,Z -23.439,A -90.000,B 90.000,C 0.000} C_DIS
LIN {X -109.246,Y -7.308,Z -23.356,A -90.000,B 90.000,C 0.000} C_DIS
LIN {X -108.843,Y -7.308,Z -23.142,A -90.000,B 90.000,C 0.000} C_DIS
LIN {X -108.715,Y -7.308,Z -23.086,A -90.000,B 90.000,C 0.000} C_DIS
LIN {X -108.439,Y -7.308,Z -22.965,A -90.000,B 90.000,C 0.000} C_DIS
LIN {X -108.211,Y -7.308,Z -22.867,A -90.000,B 90.000,C 0.000} C_DIS
LIN {X -107.806,Y -7.308,Z -22.696,A -90.000,B 90.000,C 0.000} C_DIS
LIN {X -107.436,Y -7.308,Z -22.572,A -90.000,B 90.000,C 0.000} C_DIS
LIN {X -107.074,Y -7.308,Z -22.449,A -90.000,B 90.000,C 0.000} C_DIS
LIN {X -106.848,Y -7.308,Z -22.379,A -90.000,B 90.000,C 0.000} C_DIS
LIN {X -106.653,Y -7.308,Z -22.319,A -90.000,B 90.000,C 0.000} C_DIS
LIN {X -106.345,Y -7.308,Z -22.237,A -90.000,B 90.000,C 0.000} C_DIS
LIN {X -105.845,Y -7.308,Z -22.101,A -90.000,B 90.000,C 0.000} C_DIS
LIN {X -105.614,Y -7.308,Z -22.049,A -90.000,B 90.000,C 0.000} C_DIS
LIN {X -105.283,Y -7.308,Z -21.979,A -90.000,B 90.000,C 0.000} C_DIS
LIN {X -104.901,Y -7.308,Z -21.897,A -90.000,B 90.000,C 0.000} C_DIS
LIN {X -104.570,Y -7.308,Z -21.835,A -90.000,B 90.000,C 0.000} C_DIS
LIN {X -104.430,Y -7.308,Z -21.813,A -90.000,B 90.000,C 0.000} C_DIS
LIN {X -104.151,Y -7.308,Z -21.771,A -90.000,B 90.000,C 0.000} C_DIS
LIN {X -103.770,Y -7.308,Z -21.715,A -90.000,B 90.000,C 0.000} C_DIS
LIN {X -103.677,Y -7.308,Z -21.699,A -90.000,B 90.000,C 0.000} C_DIS
LIN {X -103.573,Y -7.308,Z -21.687,A -90.000,B 90.000,C 0.000} C_DIS
LIN {X -103.214,Y -7.308,Z -21.643,A -90.000,B 90.000,C 0.000} C_DIS
LIN {X -102.480,Y -7.308,Z -21.560,A -90.000,B 90.000,C 0.000} C_DIS
LIN {X -102.343,Y -7.308,Z -21.546,A -90.000,B 90.000,C 0.000} C_DIS
LIN {X -102.080,Y -7.308,Z -21.522,A -90.000,B 90.000,C 0.000} C_DIS
LIN {X -101.933,Y -7.308,Z -21.507,A -90.000,B 90.000,C 0.000} C_DIS
LIN {X -101.774,Y -7.308,Z -21.491,A -90.000,B 90.000,C 0.000} C_DIS
LIN {X -101.668,Y -7.308,Z -21.480,A -90.000,B 90.000,C 0.000} C_DIS
LIN {X -101.655,Y -7.308,Z -21.479,A -90.000,B 90.000,C 0.000} C_DIS
LIN {X -101.620,Y -7.308,Z -21.474,A -90.000,B 90.000,C 0.000} C_DIS
LIN {X -101.575,Y -7.308,Z -21.468,A -90.000,B 90.000,C 0.000} C_DIS
LIN {X -101.513,Y -7.308,Z -21.460,A -90.000,B 90.000,C 0.000} C_DIS
LIN {X -101.508,Y -7.308,Z -21.453,A -90.000,B 90.000,C 0.000} C_DIS
LIN {X -101.507,Y -7.308,Z -21.451,A -90.000,B 90.000,C 0.000} C_DIS
LIN {X -101.506,Y -7.308,Z -21.449,A -90.000,B 90.000,C 0.000} C_DIS
LIN {X -101.498,Y -7.308,Z -21.437,A -90.000,B 90.000,C 0.000} C_DIS
LIN {X -101.497,Y -7.308,Z -21.436,A -90.000,B 90.000,C 0.000} C_DIS
LIN {X -101.495,Y -7.308,Z -21.432,A -90.000,B 90.000,C 0.000} C_DIS
LIN {X -101.460,Y -7.308,Z -21.382,A -90.000,B 90.000,C 0.000} C_DIS
LIN {X -101.459,Y -7.308,Z -21.380,A -90.000,B 90.000,C 0.000} C_DIS
LIN {X -101.388,Y -7.308,Z -21.283,A -90.000,B 90.000,C 0.000} C_DIS
LIN {X -101.173,Y -7.308,Z -20.988,A -90.000,B 90.000,C 0.000} C_DIS
LIN {X -101.084,Y -7.308,Z -20.873,A -90.000,B 90.000,C 0.000} C_DIS
LIN {X -101.061,Y -7.308,Z -20.843,A -90.000,B 90.000,C 0.000} C_DIS
LIN {X -101.045,Y -7.308,Z -20.822,A -90.000,B 90.000,C 0.000} C_DIS
LIN {X -100.962,Y -7.308,Z -20.716,A -90.000,B 90.000,C 0.000} C_DIS
LIN {X -100.897,Y -7.308,Z -20.641,A -90.000,B 90.000,C 0.000} C_DIS
LIN {X -100.848,Y -7.308,Z -20.585,A -90.000,B 90.000,C 0.000} C_DIS
LIN {X -100.720,Y -7.308,Z -20.440,A -90.000,B 90.000,C 0.000} C_DIS
LIN {X -100.523,Y -7.308,Z -20.222,A -90.000,B 90.000,C 0.000} C_DIS
LIN {X -100.434,Y -7.308,Z -20.137,A -90.000,B 90.000,C 0.000} C_DIS
LIN {X -100.314,Y -7.308,Z -20.021,A -90.000,B 90.000,C 0.000} C_DIS
LIN {X -100.248,Y -7.308,Z -19.961,A -90.000,B 90.000,C 0.000} C_DIS
LIN {X -99.955,Y -7.308,Z -19.693,A -90.000,B 90.000,C 0.000} C_DIS
LIN {X -99.858,Y -7.308,Z -19.613,A -90.000,B 90.000,C 0.000} C_DIS
LIN {X -99.290,Y -7.308,Z -19.170,A -90.000,B 90.000,C 0.000} C_DIS
LIN {X -99.278,Y -7.308,Z -19.160,A -90.000,B 90.000,C 0.000} C_DIS
LIN {X -99.270,Y -7.308,Z -19.154,A -90.000,B 90.000,C 0.000} C_DIS
LIN {X -98.887,Y -7.308,Z -18.871,A -90.000,B 90.000,C 0.000} C_DIS
LIN {X -98.624,Y -7.308,Z -18.680,A -90.000,B 90.000,C 0.000} C_DIS
LIN {X -98.471,Y -7.308,Z -18.570,A -90.000,B 90.000,C 0.000} C_DIS
LIN {X -98.285,Y -7.308,Z -18.443,A -90.000,B 90.000,C 0.000} C_DIS
LIN {X -97.932,Y -7.308,Z -18.202,A -90.000,B 90.000,C 0.000} C_DIS
LIN {X -97.756,Y -7.308,Z -18.088,A -90.000,B 90.000,C 0.000} C_DIS
LIN {X -97.215,Y -7.308,Z -17.739,A -90.000,B 90.000,C 0.000} C_DIS
LIN {X -97.074,Y -7.308,Z -17.649,A -90.000,B 90.000,C 0.000} C_DIS
LIN {X -96.917,Y -7.308,Z -17.556,A -90.000,B 90.000,C 0.000} C_DIS
LIN {X -96.656,Y -7.308,Z -17.401,A -90.000,B 90.000,C 0.000} C_DIS
LIN {X -96.483,Y -7.308,Z -17.304,A -90.000,B 90.000,C 0.000} C_DIS
LIN {X -96.009,Y -7.308,Z -17.035,A -90.000,B 90.000,C 0.000} C_DIS
LIN {X -95.981,Y -7.308,Z -17.020,A -90.000,B 90.000,C 0.000} C_DIS
LIN {X -95.969,Y -7.308,Z -17.013,A -90.000,B 90.000,C 0.000} C_DIS
LIN {X -95.537,Y -7.308,Z -16.814,A -90.000,B 90.000,C 0.000} C_DIS
LIN {X -95.528,Y -7.308,Z -16.809,A -90.000,B 90.000,C 0.000} C_DIS
LIN {X -95.024,Y -7.308,Z -16.588,A -90.000,B 90.000,C 0.000} C_DIS
LIN {X -94.756,Y -7.308,Z -16.473,A -90.000,B 90.000,C 0.000} C_DIS
LIN {X -94.526,Y -7.308,Z -16.395,A -90.000,B 90.000,C 0.000} C_DIS
LIN {X -94.296,Y -7.308,Z -16.316,A -90.000,B 90.000,C 0.000} C_DIS
LIN {X -94.181,Y -7.308,Z -16.278,A -90.000,B 90.000,C 0.000} C_DIS
LIN {X -93.765,Y -7.308,Z -16.151,A -90.000,B 90.000,C 0.000} C_DIS
LIN {X -93.454,Y -7.308,Z -16.056,A -90.000,B 90.000,C 0.000} C_DIS
LIN {X -93.295,Y -7.308,Z -16.008,A -90.000,B 90.000,C 0.000} C_DIS
LIN {X -92.951,Y -7.308,Z -15.930,A -90.000,B 90.000,C 0.000} C_DIS
LIN {X -92.819,Y -7.308,Z -15.900,A -90.000,B 90.000,C 0.000} C_DIS
LIN {X -92.341,Y -7.308,Z -15.813,A -90.000,B 90.000,C 0.000} C_DIS
LIN {X -91.887,Y -7.308,Z -15.731,A -90.000,B 90.000,C 0.000} C_DIS
LIN {X -91.757,Y -7.308,Z -15.716,A -90.000,B 90.000,C 0.000} C_DIS
LIN {X -91.403,Y -7.308,Z -15.673,A -90.000,B 90.000,C 0.000} C_DIS
LIN {X -90.755,Y -7.308,Z -15.604,A -90.000,B 90.000,C 0.000} C_DIS
LIN {X -90.382,Y -7.308,Z -15.565,A -90.000,B 90.000,C 0.000} C_DIS
LIN {X -90.346,Y -7.308,Z -15.561,A -90.000,B 90.000,C 0.000} C_DIS
LIN {X -90.345,Y -7.308,Z -15.561,A -90.000,B 90.000,C 0.000} C_DIS
LIN {X -90.310,Y -7.308,Z -15.559,A -90.000,B 90.000,C 0.000} C_DIS
LIN {X -89.566,Y -7.308,Z -15.513,A -90.000,B 90.000,C 0.000} C_DIS
LIN {X -89.550,Y -7.308,Z -15.512,A -90.000,B 90.000,C 0.000} C_DIS
LIN {X -89.450,Y -7.308,Z -15.499,A -90.000,B 90.000,C 0.000} C_DIS
LIN {X -89.154,Y -7.308,Z -15.460,A -90.000,B 90.000,C 0.000} C_DIS
LIN {X -89.152,Y -7.308,Z -15.460,A -90.000,B 90.000,C 0.000} C_DIS
LIN {X -88.887,Y -7.308,Z -15.419,A -90.000,B 90.000,C 0.000} C_DIS
LIN {X -88.516,Y -7.308,Z -15.350,A -90.000,B 90.000,C 0.000} C_DIS
LIN {X -88.080,Y -7.308,Z -15.256,A -90.000,B 90.000,C 0.000} C_DIS
LIN {X -88.030,Y -7.308,Z -15.245,A -90.000,B 90.000,C 0.000} C_DIS
LIN {X -87.716,Y -7.308,Z -15.156,A -90.000,B 90.000,C 0.000} C_DIS
LIN {X -87.312,Y -7.308,Z -15.041,A -90.000,B 90.000,C 0.000} C_DIS
LIN {X -86.953,Y -7.308,Z -14.925,A -90.000,B 90.000,C 0.000} C_DIS
LIN {X -86.912,Y -7.308,Z -14.911,A -90.000,B 90.000,C 0.000} C_DIS
LIN {X -86.875,Y -7.308,Z -14.897,A -90.000,B 90.000,C 0.000} C_DIS
LIN {X -86.804,Y -7.308,Z -14.870,A -90.000,B 90.000,C 0.000} C_DIS
LIN {X -86.714,Y -7.308,Z -14.837,A -90.000,B 90.000,C 0.000} C_DIS
LIN {X -86.591,Y -7.308,Z -14.785,A -90.000,B 90.000,C 0.000} C_DIS
LIN {X -86.404,Y -7.308,Z -14.707,A -90.000,B 90.000,C 0.000} C_DIS
LIN {X -86.158,Y -7.308,Z -14.603,A -90.000,B 90.000,C 0.000} C_DIS
LIN {X -86.085,Y -7.308,Z -14.570,A -90.000,B 90.000,C 0.000} C_DIS
LIN {X -85.996,Y -7.308,Z -14.529,A -90.000,B 90.000,C 0.000} C_DIS
LIN {X -85.805,Y -7.308,Z -14.442,A -90.000,B 90.000,C 0.000} C_DIS
LIN {X -85.591,Y -7.308,Z -14.345,A -90.000,B 90.000,C 0.000} C_DIS
LIN {X -85.554,Y -7.308,Z -14.328,A -90.000,B 90.000,C 0.000} C_DIS
LIN {X -85.552,Y -7.308,Z -14.327,A -90.000,B 90.000,C 0.000} C_DIS
LIN {X -85.549,Y -7.308,Z -14.326,A -90.000,B 90.000,C 0.000} C_DIS
LIN {X -85.490,Y -7.308,Z -14.300,A -90.000,B 90.000,C 0.000} C_DIS
LIN {X -85.291,Y -7.308,Z -14.213,A -90.000,B 90.000,C 0.000} C_DIS
LIN {X -85.013,Y -7.308,Z -14.092,A -90.000,B 90.000,C 0.000} C_DIS
LIN {X -85.008,Y -7.308,Z -14.091,A -90.000,B 90.000,C 0.000} C_DIS
LIN {X -84.910,Y -7.308,Z -14.057,A -90.000,B 90.000,C 0.000} C_DIS
LIN {X -84.823,Y -7.308,Z -14.027,A -90.000,B 90.000,C 0.000} C_DIS
LIN {X -84.814,Y -7.308,Z -14.024,A -90.000,B 90.000,C 0.000} C_DIS
LIN {X -84.609,Y -7.308,Z -13.941,A -90.000,B 90.000,C 0.000} C_DIS
LIN {X -84.318,Y -7.308,Z -13.824,A -90.000,B 90.000,C 0.000} C_DIS
LIN {X -84.311,Y -7.308,Z -13.821,A -90.000,B 90.000,C 0.000} C_DIS
LIN {X -84.195,Y -7.308,Z -13.782,A -90.000,B 90.000,C 0.000} C_DIS
LIN {X -84.071,Y -7.308,Z -13.740,A -90.000,B 90.000,C 0.000} C_DIS
LIN {X -83.852,Y -7.308,Z -13.666,A -90.000,B 90.000,C 0.000} C_DIS
LIN {X -83.848,Y -7.308,Z -13.665,A -90.000,B 90.000,C 0.000} C_DIS
LIN {X -83.844,Y -7.308,Z -13.664,A -90.000,B 90.000,C 0.000} C_DIS
LIN {X -83.748,Y -7.308,Z -13.639,A -90.000,B 90.000,C 0.000} C_DIS
LIN {X -83.644,Y -7.308,Z -13.611,A -90.000,B 90.000,C 0.000} C_DIS
LIN {X -83.636,Y -7.308,Z -13.609,A -90.000,B 90.000,C 0.000} C_DIS
LIN {X -83.509,Y -7.308,Z -13.566,A -90.000,B 90.000,C 0.000} C_DIS
LIN {X -83.463,Y -7.308,Z -13.551,A -90.000,B 90.000,C 0.000} C_DIS
LIN {X -83.441,Y -7.308,Z -13.543,A -90.000,B 90.000,C 0.000} C_DIS
LIN {X -83.033,Y -7.308,Z -13.407,A -90.000,B 90.000,C 0.000} C_DIS
LIN {X -83.032,Y -7.308,Z -13.407,A -90.000,B 90.000,C 0.000} C_DIS
LIN {X -82.990,Y -7.308,Z -13.394,A -90.000,B 90.000,C 0.000} C_DIS
LIN {X -82.940,Y -7.308,Z -13.380,A -90.000,B 90.000,C 0.000} C_DIS
LIN {X -82.838,Y -7.308,Z -13.349,A -90.000,B 90.000,C 0.000} C_DIS
LIN {X -82.837,Y -7.308,Z -13.349,A -90.000,B 90.000,C 0.000} C_DIS
LIN {X -82.723,Y -7.308,Z -13.323,A -90.000,B 90.000,C 0.000} C_DIS
LIN {X -82.362,Y -7.308,Z -13.242,A -90.000,B 90.000,C 0.000} C_DIS
LIN {X -82.360,Y -7.308,Z -13.241,A -90.000,B 90.000,C 0.000} C_DIS
LIN {X -82.357,Y -7.308,Z -13.241,A -90.000,B 90.000,C 0.000} C_DIS
LIN {X -81.920,Y -7.308,Z -13.152,A -90.000,B 90.000,C 0.000} C_DIS
LIN {X -81.692,Y -7.308,Z -13.106,A -90.000,B 90.000,C 0.000} C_DIS
LIN {X -81.659,Y -7.308,Z -13.099,A -90.000,B 90.000,C 0.000} C_DIS
LIN {X -81.654,Y -7.308,Z -13.098,A -90.000,B 90.000,C 0.000} C_DIS
LIN {X -81.645,Y -7.308,Z -13.096,A -90.000,B 90.000,C 0.000} C_DIS
LIN {X -81.386,Y -7.308,Z -13.038,A -90.000,B 90.000,C 0.000} C_DIS
LIN {X -81.385,Y -7.308,Z -13.038,A -90.000,B 90.000,C 0.000} C_DIS
LIN {X -81.378,Y -7.308,Z -13.037,A -90.000,B 90.000,C 0.000} C_DIS
LIN {X -81.302,Y -7.308,Z -13.028,A -90.000,B 90.000,C 0.000} C_DIS
LIN {X -80.901,Y -7.308,Z -12.980,A -90.000,B 90.000,C 0.000} C_DIS
LIN {X -80.900,Y -7.308,Z -12.980,A -90.000,B 90.000,C 0.000} C_DIS
LIN {X -80.790,Y -7.308,Z -12.970,A -90.000,B 90.000,C 0.000} C_DIS
LIN {X -80.783,Y -7.308,Z -12.969,A -90.000,B 90.000,C 0.000} C_DIS
LIN {X -80.119,Y -7.308,Z -12.910,A -90.000,B 90.000,C 0.000} C_DIS
LIN {X -80.101,Y -7.308,Z -12.909,A -90.000,B 90.000,C 0.000} C_DIS
LIN {X -80.004,Y -7.308,Z -12.900,A -90.000,B 90.000,C 0.000} C_DIS
LIN {X -79.939,Y -7.308,Z -12.899,A -90.000,B 90.000,C 0.000} C_DIS
LIN {X -79.793,Y -7.308,Z -12.896,A -90.000,B 90.000,C 0.000} C_DIS
LIN {X -79.533,Y -7.308,Z -12.892,A -90.000,B 90.000,C 0.000} C_DIS
LIN {X -79.519,Y -7.308,Z -12.891,A -90.000,B 90.000,C 0.000} C_DIS
LIN {X -79.517,Y -7.308,Z -12.891,A -90.000,B 90.000,C 0.000} C_DIS
LIN {X -79.512,Y -7.308,Z -12.892,A -90.000,B 90.000,C 0.000} C_DIS
LIN {X -79.114,Y -7.308,Z -12.903,A -90.000,B 90.000,C 0.000} C_DIS
LIN {X -79.050,Y -7.308,Z -12.904,A -90.000,B 90.000,C 0.000} C_DIS
LIN {X -78.615,Y -7.308,Z -12.916,A -90.000,B 90.000,C 0.000} C_DIS
LIN {X -78.592,Y -7.308,Z -12.917,A -90.000,B 90.000,C 0.000} C_DIS
LIN {X -78.528,Y -7.308,Z -12.923,A -90.000,B 90.000,C 0.000} C_DIS
LIN {X -78.381,Y -7.308,Z -12.935,A -90.000,B 90.000,C 0.000} C_DIS
LIN {X -78.228,Y -7.308,Z -12.948,A -90.000,B 90.000,C 0.000} C_DIS
LIN {X -78.110,Y -7.308,Z -12.958,A -90.000,B 90.000,C 0.000} C_DIS
LIN {X -78.106,Y -7.308,Z -12.958,A -90.000,B 90.000,C 0.000} C_DIS
LIN {X -78.104,Y -7.308,Z -12.959,A -90.000,B 90.000,C 0.000} C_DIS
LIN {X -77.981,Y -7.308,Z -12.976,A -90.000,B 90.000,C 0.000} C_DIS
LIN {X -77.950,Y -7.308,Z -12.980,A -90.000,B 90.000,C 0.000} C_DIS
LIN {X -77.888,Y -7.308,Z -12.988,A -90.000,B 90.000,C 0.000} C_DIS
LIN {X -77.884,Y -7.308,Z -12.989,A -90.000,B 90.000,C 0.000} C_DIS
LIN {X -77.477,Y -7.308,Z -13.046,A -90.000,B 90.000,C 0.000} C_DIS
LIN {X -77.321,Y -7.308,Z -13.068,A -90.000,B 90.000,C 0.000} C_DIS
LIN {X -76.988,Y -7.308,Z -13.114,A -90.000,B 90.000,C 0.000} C_DIS
LIN {X -76.919,Y -7.308,Z -13.124,A -90.000,B 90.000,C 0.000} C_DIS
LIN {X -76.848,Y -7.308,Z -13.137,A -90.000,B 90.000,C 0.000} C_DIS
LIN {X -76.749,Y -7.308,Z -13.156,A -90.000,B 90.000,C 0.000} C_DIS
LIN {X -76.656,Y -7.308,Z -13.173,A -90.000,B 90.000,C 0.000} C_DIS
LIN {X -76.443,Y -7.308,Z -13.214,A -90.000,B 90.000,C 0.000} C_DIS
LIN {X -76.440,Y -7.308,Z -13.215,A -90.000,B 90.000,C 0.000} C_DIS
LIN {X -76.433,Y -7.308,Z -13.216,A -90.000,B 90.000,C 0.000} C_DIS
LIN {X -75.926,Y -7.308,Z -13.350,A -90.000,B 90.000,C 0.000} C_DIS
LIN {X -75.571,Y -7.308,Z -13.444,A -90.000,B 90.000,C 0.000} C_DIS
LIN {X -75.531,Y -7.308,Z -13.449,A -90.000,B 90.000,C 0.000} C_DIS
LIN {X -75.526,Y -7.308,Z -13.450,A -90.000,B 90.000,C 0.000} C_DIS
LIN {X -75.249,Y -7.308,Z -13.489,A -90.000,B 90.000,C 0.000} C_DIS
LIN {X -75.246,Y -7.308,Z -13.490,A -90.000,B 90.000,C 0.000} C_DIS
LIN {X -75.242,Y -7.308,Z -13.490,A -90.000,B 90.000,C 0.000} C_DIS
LIN {X -74.948,Y -7.308,Z -13.529,A -90.000,B 90.000,C 0.000} C_DIS
LIN {X -74.932,Y -7.308,Z -13.531,A -90.000,B 90.000,C 0.000} C_DIS
LIN {X -74.627,Y -7.308,Z -13.578,A -90.000,B 90.000,C 0.000} C_DIS
LIN {X -74.497,Y -7.308,Z -13.598,A -90.000,B 90.000,C 0.000} C_DIS
LIN {X -74.270,Y -7.308,Z -13.642,A -90.000,B 90.000,C 0.000} C_DIS
LIN {X -74.151,Y -7.308,Z -13.665,A -90.000,B 90.000,C 0.000} C_DIS
LIN {X -74.145,Y -7.308,Z -13.666,A -90.000,B 90.000,C 0.000} C_DIS
LIN {X -73.965,Y -7.308,Z -13.701,A -90.000,B 90.000,C 0.000} C_DIS
LIN {X -73.577,Y -7.308,Z -13.777,A -90.000,B 90.000,C 0.000} C_DIS
LIN {X -73.182,Y -7.308,Z -13.862,A -90.000,B 90.000,C 0.000} C_DIS
LIN {X -73.146,Y -7.308,Z -13.870,A -90.000,B 90.000,C 0.000} C_DIS
LIN {X -73.098,Y -7.308,Z -13.881,A -90.000,B 90.000,C 0.000} C_DIS
LIN {X -73.091,Y -7.308,Z -13.882,A -90.000,B 90.000,C 0.000} C_DIS
LIN {X -73.073,Y -7.308,Z -13.886,A -90.000,B 90.000,C 0.000} C_DIS
LIN {X -73.012,Y -7.308,Z -13.900,A -90.000,B 90.000,C 0.000} C_DIS
LIN {X -72.427,Y -7.308,Z -14.034,A -90.000,B 90.000,C 0.000} C_DIS
LIN {X -72.425,Y -7.308,Z -14.035,A -90.000,B 90.000,C 0.000} C_DIS
LIN {X -72.352,Y -7.308,Z -14.055,A -90.000,B 90.000,C 0.000} C_DIS
LIN {X -72.329,Y -7.308,Z -14.061,A -90.000,B 90.000,C 0.000} C_DIS
LIN {X -72.286,Y -7.308,Z -14.073,A -90.000,B 90.000,C 0.000} C_DIS
LIN {X -71.907,Y -7.308,Z -14.156,A -90.000,B 90.000,C 0.000} C_DIS
LIN {X -71.712,Y -7.308,Z -14.198,A -90.000,B 90.000,C 0.000} C_DIS
LIN {X -71.555,Y -7.308,Z -14.232,A -90.000,B 90.000,C 0.000} C_DIS
LIN {X -71.015,Y -7.308,Z -14.319,A -90.000,B 90.000,C 0.000} C_DIS
LIN {X -70.678,Y -7.308,Z -14.373,A -90.000,B 90.000,C 0.000} C_DIS
LIN {X -70.504,Y -7.308,Z -14.386,A -90.000,B 90.000,C 0.000} C_DIS
LIN {X -70.474,Y -7.308,Z -14.388,A -90.000,B 90.000,C 0.000} C_DIS
LIN {X -70.219,Y -7.308,Z -14.406,A -90.000,B 90.000,C 0.000} C_DIS
LIN {X -70.122,Y -7.308,Z -14.414,A -90.000,B 90.000,C 0.000} C_DIS
LIN {X -69.526,Y -7.308,Z -14.460,A -90.000,B 90.000,C 0.000} C_DIS
LIN {X -69.048,Y -7.308,Z -14.474,A -90.000,B 90.000,C 0.000} C_DIS
LIN {X -68.538,Y -7.308,Z -14.490,A -90.000,B 90.000,C 0.000} C_DIS
LIN {X -67.983,Y -7.308,Z -14.511,A -90.000,B 90.000,C 0.000} C_DIS
LIN {X -66.592,Y -7.308,Z -14.544,A -90.000,B 90.000,C 0.000} C_DIS
LIN {X -66.525,Y -7.308,Z -14.546,A -90.000,B 90.000,C 0.000} C_DIS
LIN {X -66.324,Y -7.308,Z -14.556,A -90.000,B 90.000,C 0.000} C_DIS
LIN {X -65.216,Y -7.308,Z -14.622,A -90.000,B 90.000,C 0.000} C_DIS
LIN {X -65.076,Y -7.308,Z -14.635,A -90.000,B 90.000,C 0.000} C_DIS
LIN {X -64.443,Y -7.308,Z -14.716,A -90.000,B 90.000,C 0.000} C_DIS
LIN {X -63.743,Y -7.308,Z -14.805,A -90.000,B 90.000,C 0.000} C_DIS
LIN {X -63.596,Y -7.308,Z -14.826,A -90.000,B 90.000,C 0.000} C_DIS
LIN {X -62.633,Y -7.308,Z -14.994,A -90.000,B 90.000,C 0.000} C_DIS
LIN {X -62.461,Y -7.308,Z -15.024,A -90.000,B 90.000,C 0.000} C_DIS
LIN {X -62.009,Y -7.308,Z -15.111,A -90.000,B 90.000,C 0.000} C_DIS
LIN {X -61.344,Y -7.308,Z -15.250,A -90.000,B 90.000,C 0.000} C_DIS
LIN {X -61.125,Y -7.308,Z -15.293,A -90.000,B 90.000,C 0.000} C_DIS
LIN {X -60.233,Y -7.308,Z -15.470,A -90.000,B 90.000,C 0.000} C_DIS
LIN {X -59.746,Y -7.308,Z -15.546,A -90.000,B 90.000,C 0.000} C_DIS
LIN {X -59.492,Y -7.308,Z -15.585,A -90.000,B 90.000,C 0.000} C_DIS
LIN {X -59.136,Y -7.308,Z -15.633,A -90.000,B 90.000,C 0.000} C_DIS
LIN {X -59.132,Y -7.308,Z -15.633,A -90.000,B 90.000,C 0.000} C_DIS
LIN {X -58.963,Y -7.308,Z -15.659,A -90.000,B 90.000,C 0.000} C_DIS
LIN {X -58.700,Y -7.308,Z -15.700,A -90.000,B 90.000,C 0.000} C_DIS
LIN {X -58.149,Y -7.308,Z -15.786,A -90.000,B 90.000,C 0.000} C_DIS
LIN {X -57.763,Y -7.308,Z -15.848,A -90.000,B 90.000,C 0.000} C_DIS
LIN {X -57.153,Y -7.308,Z -15.945,A -90.000,B 90.000,C 0.000} C_DIS
LIN {X -56.145,Y -7.308,Z -16.132,A -90.000,B 90.000,C 0.000} C_DIS
LIN {X -56.003,Y -7.308,Z -16.158,A -90.000,B 90.000,C 0.000} C_DIS
LIN {X -55.595,Y -7.308,Z -16.240,A -90.000,B 90.000,C 0.000} C_DIS
LIN {X -54.787,Y -7.308,Z -16.415,A -90.000,B 90.000,C 0.000} C_DIS
LIN {X -54.180,Y -7.308,Z -16.551,A -90.000,B 90.000,C 0.000} C_DIS
LIN {X -54.151,Y -7.308,Z -16.558,A -90.000,B 90.000,C 0.000} C_DIS
LIN {X -54.021,Y -7.308,Z -16.589,A -90.000,B 90.000,C 0.000} C_DIS
LIN {X -52.425,Y -7.308,Z -16.971,A -90.000,B 90.000,C 0.000} C_DIS
LIN {X -51.849,Y -7.308,Z -17.114,A -90.000,B 90.000,C 0.000} C_DIS
LIN {X -50.300,Y -7.308,Z -17.497,A -90.000,B 90.000,C 0.000} C_DIS
LIN {X -47.958,Y -7.308,Z -18.085,A -90.000,B 90.000,C 0.000} C_DIS
LIN {X -47.662,Y -7.308,Z -18.159,A -90.000,B 90.000,C 0.000} C_DIS
LIN {X -46.877,Y -7.308,Z -18.353,A -90.000,B 90.000,C 0.000} C_DIS
LIN {X -46.521,Y -7.308,Z -18.440,A -90.000,B 90.000,C 0.000} C_DIS
LIN {X -44.746,Y -7.308,Z -18.884,A -90.000,B 90.000,C 0.000} C_DIS
LIN {X -41.859,Y -7.308,Z -19.528,A -90.000,B 90.000,C 0.000} C_DIS
LIN {X -41.335,Y -7.308,Z -19.655,A -90.000,B 90.000,C 0.000} C_DIS
LIN {X -40.214,Y -7.308,Z -19.893,A -90.000,B 90.000,C 0.000} C_DIS
LIN {X -39.785,Y -7.308,Z -19.988,A -90.000,B 90.000,C 0.000} C_DIS
LIN {X -39.603,Y -7.308,Z -20.028,A -90.000,B 90.000,C 0.000} C_DIS
LIN {X -37.961,Y -7.308,Z -20.391,A -90.000,B 90.000,C 0.000} C_DIS
LIN {X -37.688,Y -7.308,Z -20.445,A -90.000,B 90.000,C 0.000} C_DIS
LIN {X -37.612,Y -7.308,Z -20.459,A -90.000,B 90.000,C 0.000} C_DIS
LIN {X -37.539,Y -7.308,Z -20.474,A -90.000,B 90.000,C 0.000} C_DIS
LIN {X -37.190,Y -7.308,Z -20.544,A -90.000,B 90.000,C 0.000} C_DIS
LIN {X -37.092,Y -7.308,Z -20.564,A -90.000,B 90.000,C 0.000} C_DIS
LIN {X -34.474,Y -7.308,Z -21.130,A -90.000,B 90.000,C 0.000} C_DIS
LIN {X -33.029,Y -7.308,Z -21.424,A -90.000,B 90.000,C 0.000} C_DIS
LIN {X -31.502,Y -7.308,Z -21.759,A -90.000,B 90.000,C 0.000} C_DIS
LIN {X -29.687,Y -7.308,Z -22.147,A -90.000,B 90.000,C 0.000} C_DIS
LIN {X -28.828,Y -7.308,Z -22.340,A -90.000,B 90.000,C 0.000} C_DIS
LIN {X -26.779,Y -7.308,Z -22.797,A -90.000,B 90.000,C 0.000} C_DIS
LIN {X -26.362,Y -7.308,Z -22.892,A -90.000,B 90.000,C 0.000} C_DIS
LIN {X -24.102,Y -7.308,Z -23.408,A -90.000,B 90.000,C 0.000} C_DIS
LIN {X -24.017,Y -7.308,Z -23.428,A -90.000,B 90.000,C 0.000} C_DIS
LIN {X -24.013,Y -7.308,Z -23.429,A -90.000,B 90.000,C 0.000} C_DIS
LIN {X -23.361,Y -7.308,Z -23.577,A -90.000,B 90.000,C 0.000} C_DIS
LIN {X -21.872,Y -7.308,Z -23.929,A -90.000,B 90.000,C 0.000} C_DIS
LIN {X -21.710,Y -7.308,Z -23.966,A -90.000,B 90.000,C 0.000} C_DIS
LIN {X -19.778,Y -7.308,Z -24.421,A -90.000,B 90.000,C 0.000} C_DIS
LIN {X -19.378,Y -7.308,Z -24.513,A -90.000,B 90.000,C 0.000} C_DIS
LIN {X -17.636,Y -7.308,Z -24.924,A -90.000,B 90.000,C 0.000} C_DIS
LIN {X -16.955,Y -7.308,Z -25.082,A -90.000,B 90.000,C 0.000} C_DIS
LIN {X -15.411,Y -7.308,Z -25.447,A -90.000,B 90.000,C 0.000} C_DIS
LIN {X -14.374,Y -7.308,Z -25.692,A -90.000,B 90.000,C 0.000} C_DIS
LIN {X -12.856,Y -7.308,Z -26.059,A -90.000,B 90.000,C 0.000} C_DIS
LIN {X -11.563,Y -7.308,Z -26.366,A -90.000,B 90.000,C 0.000} C_DIS
LIN {X -9.348,Y -7.308,Z -26.894,A -90.000,B 90.000,C 0.000} C_DIS
LIN {X -8.588,Y -7.308,Z -27.072,A -90.000,B 90.000,C 0.000} C_DIS
LIN {X -5.616,Y -7.308,Z -27.750,A -90.000,B 90.000,C 0.000} C_DIS
LIN {X -5.521,Y -7.308,Z -27.771,A -90.000,B 90.000,C 0.000} C_DIS
LIN {X -5.179,Y -7.308,Z -27.843,A -90.000,B 90.000,C 0.000} C_DIS
LIN {X -5.157,Y -7.308,Z -27.848,A -90.000,B 90.000,C 0.000} C_DIS
LIN {X -5.123,Y -7.308,Z -27.855,A -90.000,B 90.000,C 0.000} C_DIS
LIN {X -2.725,Y -7.308,Z -28.373,A -90.000,B 90.000,C 0.000} C_DIS
LIN {X -2.133,Y -7.308,Z -28.485,A -90.000,B 90.000,C 0.000} C_DIS
LIN {X -0.152,Y -7.308,Z -28.888,A -90.000,B 90.000,C 0.000} C_DIS
LIN {X 0.278,Y -7.308,Z -28.975,A -90.000,B 90.000,C 0.000} C_DIS
LIN {X 2.269,Y -7.308,Z -29.352,A -90.000,B 90.000,C 0.000} C_DIS
LIN {X 3.186,Y -7.308,Z -29.518,A -90.000,B 90.000,C 0.000} C_DIS
LIN {X 4.600,Y -7.308,Z -29.784,A -90.000,B 90.000,C 0.000} C_DIS
LIN {X 5.909,Y -7.308,Z -30.006,A -90.000,B 90.000,C 0.000} C_DIS
LIN {X 6.804,Y -7.308,Z -30.185,A -90.000,B 90.000,C 0.000} C_DIS
LIN {X 8.374,Y -7.308,Z -30.456,A -90.000,B 90.000,C 0.000} C_DIS
LIN {X 10.305,Y -7.308,Z -30.842,A -90.000,B 90.000,C 0.000} C_DIS
LIN {X 10.367,Y -7.308,Z -30.856,A -90.000,B 90.000,C 0.000} C_DIS
LIN {X 10.531,Y -7.308,Z -30.893,A -90.000,B 90.000,C 0.000} C_DIS
LIN {X 11.573,Y -7.308,Z -31.113,A -90.000,B 90.000,C 0.000} C_DIS
LIN {X 12.407,Y -7.308,Z -31.302,A -90.000,B 90.000,C 0.000} C_DIS
LIN {X 13.224,Y -7.308,Z -31.485,A -90.000,B 90.000,C 0.000} C_DIS
LIN {X 14.180,Y -7.308,Z -31.699,A -90.000,B 90.000,C 0.000} C_DIS
LIN {X 15.435,Y -7.308,Z -31.948,A -90.000,B 90.000,C 0.000} C_DIS
LIN {X 15.824,Y -7.308,Z -32.027,A -90.000,B 90.000,C 0.000} C_DIS
LIN {X 16.794,Y -7.308,Z -32.175,A -90.000,B 90.000,C 0.000} C_DIS
LIN {X 16.810,Y -7.308,Z -32.178,A -90.000,B 90.000,C 0.000} C_DIS
LIN {X 17.137,Y -7.308,Z -32.228,A -90.000,B 90.000,C 0.000} C_DIS
LIN {X 17.300,Y -7.308,Z -32.248,A -90.000,B 90.000,C 0.000} C_DIS
LIN {X 17.445,Y -7.308,Z -32.266,A -90.000,B 90.000,C 0.000} C_DIS
LIN {X 18.245,Y -7.308,Z -32.362,A -90.000,B 90.000,C 0.000} C_DIS
LIN {X 18.691,Y -7.308,Z -32.430,A -90.000,B 90.000,C 0.000} C_DIS
LIN {X 20.176,Y -7.308,Z -32.588,A -90.000,B 90.000,C 0.000} C_DIS
LIN {X 20.295,Y -7.308,Z -32.601,A -90.000,B 90.000,C 0.000} C_DIS
LIN {X 20.542,Y -7.308,Z -32.628,A -90.000,B 90.000,C 0.000} C_DIS
LIN {X 21.382,Y -7.308,Z -32.726,A -90.000,B 90.000,C 0.000} C_DIS
LIN {X 21.450,Y -7.308,Z -32.734,A -90.000,B 90.000,C 0.000} C_DIS
LIN {X 21.665,Y -7.308,Z -32.759,A -90.000,B 90.000,C 0.000} C_DIS
LIN {X 21.835,Y -7.308,Z -32.781,A -90.000,B 90.000,C 0.000} C_DIS
LIN {X 22.539,Y -7.308,Z -32.881,A -90.000,B 90.000,C 0.000} C_DIS
LIN {X 23.299,Y -7.308,Z -32.989,A -90.000,B 90.000,C 0.000} C_DIS
LIN {X 24.131,Y -7.308,Z -33.130,A -90.000,B 90.000,C 0.000} C_DIS
LIN {X 24.406,Y -7.308,Z -33.181,A -90.000,B 90.000,C 0.000} C_DIS
LIN {X 24.610,Y -7.308,Z -33.219,A -90.000,B 90.000,C 0.000} C_DIS
LIN {X 25.107,Y -7.308,Z -33.312,A -90.000,B 90.000,C 0.000} C_DIS
LIN {X 25.217,Y -7.308,Z -33.333,A -90.000,B 90.000,C 0.000} C_DIS
LIN {X 26.268,Y -7.308,Z -33.566,A -90.000,B 90.000,C 0.000} C_DIS
LIN {X 26.683,Y -7.308,Z -33.655,A -90.000,B 90.000,C 0.000} C_DIS
LIN {X 27.456,Y -7.308,Z -33.848,A -90.000,B 90.000,C 0.000} C_DIS
LIN {X 28.243,Y -7.308,Z -34.042,A -90.000,B 90.000,C 0.000} C_DIS
LIN {X 28.533,Y -7.308,Z -34.123,A -90.000,B 90.000,C 0.000} C_DIS
LIN {X 29.669,Y -7.308,Z -34.441,A -90.000,B 90.000,C 0.000} C_DIS
LIN {X 29.834,Y -7.308,Z -34.486,A -90.000,B 90.000,C 0.000} C_DIS
LIN {X 29.965,Y -7.308,Z -34.522,A -90.000,B 90.000,C 0.000} C_DIS
LIN {X 30.110,Y -7.308,Z -34.565,A -90.000,B 90.000,C 0.000} C_DIS
LIN {X 30.416,Y -7.308,Z -34.656,A -90.000,B 90.000,C 0.000} C_DIS
LIN {X 30.424,Y -7.308,Z -34.659,A -90.000,B 90.000,C 0.000} C_DIS
LIN {X 30.610,Y -7.308,Z -34.716,A -90.000,B 90.000,C 0.000} C_DIS
LIN {X 31.121,Y -7.308,Z -34.872,A -90.000,B 90.000,C 0.000} C_DIS
LIN {X 31.366,Y -7.308,Z -34.947,A -90.000,B 90.000,C 0.000} C_DIS
LIN {X 31.961,Y -7.308,Z -35.130,A -90.000,B 90.000,C 0.000} C_DIS
LIN {X 32.308,Y -7.308,Z -35.233,A -90.000,B 90.000,C 0.000} C_DIS
LIN {X 32.857,Y -7.308,Z -35.414,A -90.000,B 90.000,C 0.000} C_DIS
LIN {X 33.937,Y -7.308,Z -35.775,A -90.000,B 90.000,C 0.000} C_DIS
LIN {X 33.980,Y -7.308,Z -35.790,A -90.000,B 90.000,C 0.000} C_DIS
LIN {X 34.238,Y -7.308,Z -35.871,A -90.000,B 90.000,C 0.000} C_DIS
LIN {X 34.326,Y -7.308,Z -35.898,A -90.000,B 90.000,C 0.000} C_DIS
LIN {X 34.335,Y -7.308,Z -35.901,A -90.000,B 90.000,C 0.000} C_DIS
LIN {X 34.350,Y -7.308,Z -35.906,A -90.000,B 90.000,C 0.000} C_DIS
LIN {X 34.444,Y -7.308,Z -35.936,A -90.000,B 90.000,C 0.000} C_DIS
LIN {X 34.754,Y -7.308,Z -36.035,A -90.000,B 90.000,C 0.000} C_DIS
LIN {X 34.875,Y -7.308,Z -36.074,A -90.000,B 90.000,C 0.000} C_DIS
LIN {X 36.527,Y -7.308,Z -36.603,A -90.000,B 90.000,C 0.000} C_DIS
LIN {X 36.549,Y -7.308,Z -36.610,A -90.000,B 90.000,C 0.000} C_DIS
LIN {X 36.585,Y -7.308,Z -36.622,A -90.000,B 90.000,C 0.000} C_DIS
LIN {X 37.308,Y -7.308,Z -36.855,A -90.000,B 90.000,C 0.000} C_DIS
LIN {X 38.942,Y -7.308,Z -37.383,A -90.000,B 90.000,C 0.000} C_DIS
LIN {X 38.963,Y -7.308,Z -37.390,A -90.000,B 90.000,C 0.000} C_DIS
LIN {X 39.012,Y -7.308,Z -37.406,A -90.000,B 90.000,C 0.000} C_DIS
LIN {X 39.154,Y -7.308,Z -37.454,A -90.000,B 90.000,C 0.000} C_DIS
LIN {X 39.464,Y -7.308,Z -37.560,A -90.000,B 90.000,C 0.000} C_DIS
LIN {X 40.222,Y -7.308,Z -37.787,A -90.000,B 90.000,C 0.000} C_DIS
LIN {X 41.425,Y -7.308,Z -38.147,A -90.000,B 90.000,C 0.000} C_DIS
LIN {X 41.517,Y -7.308,Z -38.178,A -90.000,B 90.000,C 0.000} C_DIS
LIN {X 41.621,Y -7.308,Z -38.212,A -90.000,B 90.000,C 0.000} C_DIS
LIN {X 41.797,Y -7.308,Z -38.271,A -90.000,B 90.000,C 0.000} C_DIS
LIN {X 42.371,Y -7.308,Z -38.461,A -90.000,B 90.000,C 0.000} C_DIS
LIN {X 42.474,Y -7.308,Z -38.496,A -90.000,B 90.000,C 0.000} C_DIS
LIN {X 42.646,Y -7.308,Z -38.553,A -90.000,B 90.000,C 0.000} C_DIS
LIN {X 43.066,Y -7.308,Z -38.675,A -90.000,B 90.000,C 0.000} C_DIS
LIN {X 43.430,Y -7.308,Z -38.780,A -90.000,B 90.000,C 0.000} C_DIS
LIN {X 43.454,Y -7.308,Z -38.787,A -90.000,B 90.000,C 0.000} C_DIS
LIN {X 43.658,Y -7.308,Z -38.848,A -90.000,B 90.000,C 0.000} C_DIS
LIN {X 43.716,Y -7.308,Z -38.866,A -90.000,B 90.000,C 0.000} C_DIS
LIN {X 43.897,Y -7.308,Z -38.920,A -90.000,B 90.000,C 0.000} C_DIS
LIN {X 44.037,Y -7.308,Z -38.969,A -90.000,B 90.000,C 0.000} C_DIS
LIN {X 44.832,Y -7.308,Z -39.248,A -90.000,B 90.000,C 0.000} C_DIS
LIN {X 45.492,Y -7.308,Z -39.480,A -90.000,B 90.000,C 0.000} C_DIS
LIN {X 46.517,Y -7.308,Z -39.840,A -90.000,B 90.000,C 0.000} C_DIS
LIN {X 46.609,Y -7.308,Z -39.873,A -90.000,B 90.000,C 0.000} C_DIS
LIN {X 46.877,Y -7.308,Z -39.984,A -90.000,B 90.000,C 0.000} C_DIS
LIN {X 47.034,Y -7.308,Z -40.048,A -90.000,B 90.000,C 0.000} C_DIS
LIN {X 47.060,Y -7.308,Z -40.059,A -90.000,B 90.000,C 0.000} C_DIS
LIN {X 47.204,Y -7.308,Z -40.122,A -90.000,B 90.000,C 0.000} C_DIS
LIN {X 47.721,Y -7.308,Z -40.346,A -90.000,B 90.000,C 0.000} C_DIS
LIN {X 48.446,Y -7.308,Z -40.662,A -90.000,B 90.000,C 0.000} C_DIS
LIN {X 49.202,Y -7.308,Z -40.991,A -90.000,B 90.000,C 0.000} C_DIS
LIN {X 49.338,Y -7.308,Z -41.050,A -90.000,B 90.000,C 0.000} C_DIS
LIN {X 49.484,Y -7.308,Z -41.114,A -90.000,B 90.000,C 0.000} C_DIS
LIN {X 49.502,Y -7.308,Z -41.123,A -90.000,B 90.000,C 0.000} C_DIS
LIN {X 49.521,Y -7.308,Z -41.132,A -90.000,B 90.000,C 0.000} C_DIS
LIN {X 49.657,Y -7.308,Z -41.202,A -90.000,B 90.000,C 0.000} C_DIS
LIN {X 49.716,Y -7.308,Z -41.231,A -90.000,B 90.000,C 0.000} C_DIS
LIN {X 49.872,Y -7.308,Z -41.314,A -90.000,B 90.000,C 0.000} C_DIS
LIN {X 50.374,Y -7.308,Z -41.581,A -90.000,B 90.000,C 0.000} C_DIS
LIN {X 51.522,Y -7.308,Z -42.190,A -90.000,B 90.000,C 0.000} C_DIS
LIN {X 52.060,Y -7.308,Z -42.475,A -90.000,B 90.000,C 0.000} C_DIS
LIN {X 52.097,Y -7.308,Z -42.495,A -90.000,B 90.000,C 0.000} C_DIS
LIN {X 52.111,Y -7.308,Z -42.503,A -90.000,B 90.000,C 0.000} C_DIS
LIN {X 52.413,Y -7.308,Z -42.666,A -90.000,B 90.000,C 0.000} C_DIS
LIN {X 52.489,Y -7.308,Z -42.707,A -90.000,B 90.000,C 0.000} C_DIS
LIN {X 52.507,Y -7.308,Z -42.717,A -90.000,B 90.000,C 0.000} C_DIS
LIN {X 52.662,Y -7.308,Z -42.803,A -90.000,B 90.000,C 0.000} C_DIS
LIN {X 52.699,Y -7.308,Z -42.823,A -90.000,B 90.000,C 0.000} C_DIS
LIN {X 52.713,Y -7.308,Z -42.832,A -90.000,B 90.000,C 0.000} C_DIS
LIN {X 52.874,Y -7.308,Z -42.934,A -90.000,B 90.000,C 0.000} C_DIS
LIN {X 54.527,Y -7.308,Z -43.976,A -90.000,B 90.000,C 0.000} C_DIS
LIN {X 54.787,Y -7.308,Z -44.140,A -90.000,B 90.000,C 0.000} C_DIS
LIN {X 55.104,Y -7.308,Z -44.340,A -90.000,B 90.000,C 0.000} C_DIS
LIN {X 55.136,Y -7.308,Z -44.362,A -90.000,B 90.000,C 0.000} C_DIS
LIN {X 55.482,Y -7.308,Z -44.597,A -90.000,B 90.000,C 0.000} C_DIS
LIN {X 55.508,Y -7.308,Z -44.614,A -90.000,B 90.000,C 0.000} C_DIS
LIN {X 55.684,Y -7.308,Z -44.745,A -90.000,B 90.000,C 0.000} C_DIS
LIN {X 56.133,Y -7.308,Z -45.079,A -90.000,B 90.000,C 0.000} C_DIS
LIN {X 56.386,Y -7.308,Z -45.266,A -90.000,B 90.000,C 0.000} C_DIS
LIN {X 57.536,Y -7.308,Z -45.807,A -90.000,B 90.000,C 0.000} C_DIS
LIN {X 57.593,Y -7.308,Z -45.836,A -90.000,B 90.000,C 0.000} C_DIS
LIN {X 57.710,Y -7.308,Z -45.896,A -90.000,B 90.000,C 0.000} C_DIS
LIN {X 57.924,Y -7.308,Z -46.004,A -90.000,B 90.000,C 0.000} C_DIS
LIN {X 57.959,Y -7.308,Z -46.022,A -90.000,B 90.000,C 0.000} C_DIS
LIN {X 57.961,Y -7.308,Z -46.022,A -90.000,B 90.000,C 0.000} C_DIS
LIN {X 59.625,Y -7.308,Z -46.878,A -90.000,B 90.000,C 0.000} C_DIS
LIN {X 59.691,Y -7.308,Z -46.910,A -90.000,B 90.000,C 0.000} C_DIS
LIN {X 60.190,Y -7.308,Z -47.156,A -90.000,B 90.000,C 0.000} C_DIS
LIN {X 60.289,Y -7.308,Z -47.206,A -90.000,B 90.000,C 0.000} C_DIS
LIN {X 60.315,Y -7.308,Z -47.219,A -90.000,B 90.000,C 0.000} C_DIS
LIN {X 60.524,Y -7.308,Z -47.325,A -90.000,B 90.000,C 0.000} C_DIS
LIN {X 60.593,Y -7.308,Z -47.360,A -90.000,B 90.000,C 0.000} C_DIS
LIN {X 60.615,Y -7.308,Z -47.371,A -90.000,B 90.000,C 0.000} C_DIS
LIN {X 61.409,Y -7.308,Z -47.788,A -90.000,B 90.000,C 0.000} C_DIS
LIN {X 61.417,Y -7.308,Z -47.792,A -90.000,B 90.000,C 0.000} C_DIS
LIN {X 61.533,Y -7.308,Z -47.850,A -90.000,B 90.000,C 0.000} C_DIS
LIN {X 62.150,Y -7.308,Z -48.155,A -90.000,B 90.000,C 0.000} C_DIS
LIN {X 62.397,Y -7.308,Z -48.280,A -90.000,B 90.000,C 0.000} C_DIS
LIN {X 62.426,Y -7.308,Z -48.294,A -90.000,B 90.000,C 0.000} C_DIS
LIN {X 62.926,Y -7.308,Z -48.548,A -90.000,B 90.000,C 0.000} C_DIS
LIN {X 63.007,Y -7.308,Z -48.590,A -90.000,B 90.000,C 0.000} C_DIS
LIN {X 63.014,Y -7.308,Z -48.593,A -90.000,B 90.000,C 0.000} C_DIS
LIN {X 63.532,Y -7.308,Z -48.861,A -90.000,B 90.000,C 0.000} C_DIS
LIN {X 63.647,Y -7.308,Z -48.920,A -90.000,B 90.000,C 0.000} C_DIS
LIN {X 64.350,Y -7.308,Z -49.281,A -90.000,B 90.000,C 0.000} C_DIS
LIN {X 64.839,Y -7.308,Z -49.524,A -90.000,B 90.000,C 0.000} C_DIS
LIN {X 65.093,Y -7.308,Z -49.651,A -90.000,B 90.000,C 0.000} C_DIS
LIN {X 65.197,Y -7.308,Z -49.706,A -90.000,B 90.000,C 0.000} C_DIS
LIN {X 65.520,Y -7.308,Z -49.876,A -90.000,B 90.000,C 0.000} C_DIS
LIN {X 66.626,Y -7.308,Z -50.463,A -90.000,B 90.000,C 0.000} C_DIS
LIN {X 67.517,Y -7.308,Z -50.937,A -90.000,B 90.000,C 0.000} C_DIS
LIN {X 67.967,Y -7.308,Z -51.199,A -90.000,B 90.000,C 0.000} C_DIS
LIN {X 69.527,Y -7.308,Z -52.102,A -90.000,B 90.000,C 0.000} C_DIS
LIN {X 69.609,Y -7.308,Z -52.152,A -90.000,B 90.000,C 0.000} C_DIS
LIN {X 71.651,Y -7.308,Z -53.398,A -90.000,B 90.000,C 0.000} C_DIS
LIN {X 71.678,Y -7.308,Z -53.416,A -90.000,B 90.000,C 0.000} C_DIS
LIN {X 73.835,Y -7.308,Z -54.782,A -90.000,B 90.000,C 0.000} C_DIS
LIN {X 74.027,Y -7.308,Z -54.907,A -90.000,B 90.000,C 0.000} C_DIS
LIN {X 75.929,Y -7.308,Z -56.143,A -90.000,B 90.000,C 0.000} C_DIS
LIN {X 76.320,Y -7.308,Z -56.399,A -90.000,B 90.000,C 0.000} C_DIS
LIN {X 77.775,Y -7.308,Z -57.362,A -90.000,B 90.000,C 0.000} C_DIS
LIN {X 78.063,Y -7.308,Z -57.553,A -90.000,B 90.000,C 0.000} C_DIS
LIN {X 78.177,Y -7.308,Z -57.629,A -90.000,B 90.000,C 0.000} C_DIS
LIN {X 78.695,Y -7.308,Z -57.980,A -90.000,B 90.000,C 0.000} C_DIS
LIN {X 79.209,Y -7.308,Z -58.337,A -90.000,B 90.000,C 0.000} C_DIS
LIN {X 79.209,Y -60.000,Z -58.337,A -90.000,B 90.000,C 0.000} C_DIS
LIN {X 103.207,Y -60.000,Z -88.531,A -90.000,B 90.000,C 0.000} C_DIS
LIN {X 103.207,Y -7.308,Z -88.531,A -90.000,B 90.000,C 0.000} C_DIS
LIN {X 103.293,Y -7.308,Z -88.699,A -90.000,B 90.000,C 0.000} C_DIS
LIN {X 103.736,Y -7.308,Z -89.585,A -90.000,B 90.000,C 0.000} C_DIS
LIN {X 103.916,Y -7.308,Z -89.979,A -90.000,B 90.000,C 0.000} C_DIS
LIN {X 104.290,Y -7.308,Z -90.831,A -90.000,B 90.000,C 0.000} C_DIS
LIN {X 104.343,Y -7.308,Z -90.969,A -90.000,B 90.000,C 0.000} C_DIS
LIN {X 104.456,Y -7.308,Z -91.264,A -90.000,B 90.000,C 0.000} C_DIS
LIN {X 104.461,Y -7.308,Z -91.275,A -90.000,B 90.000,C 0.000} C_DIS
LIN {X 104.465,Y -7.308,Z -91.285,A -90.000,B 90.000,C 0.000} C_DIS
LIN {X 104.488,Y -7.308,Z -91.349,A -90.000,B 90.000,C 0.000} C_DIS
LIN {X 104.709,Y -7.308,Z -91.939,A -90.000,B 90.000,C 0.000} C_DIS
LIN {X 104.712,Y -7.308,Z -91.949,A -90.000,B 90.000,C 0.000} C_DIS
LIN {X 104.762,Y -7.308,Z -92.079,A -90.000,B 90.000,C 0.000} C_DIS
LIN {X 104.792,Y -7.308,Z -92.157,A -90.000,B 90.000,C 0.000} C_DIS
LIN {X 104.889,Y -7.308,Z -92.409,A -90.000,B 90.000,C 0.000} C_DIS
LIN {X 104.915,Y -7.308,Z -92.493,A -90.000,B 90.000,C 0.000} C_DIS
LIN {X 105.090,Y -7.308,Z -93.058,A -90.000,B 90.000,C 0.000} C_DIS
LIN {X 105.214,Y -7.308,Z -93.440,A -90.000,B 90.000,C 0.000} C_DIS
LIN {X 105.227,Y -7.308,Z -93.480,A -90.000,B 90.000,C 0.000} C_DIS
LIN {X 105.285,Y -7.308,Z -93.698,A -90.000,B 90.000,C 0.000} C_DIS
LIN {X 105.328,Y -7.308,Z -93.857,A -90.000,B 90.000,C 0.000} C_DIS
LIN {X 105.351,Y -7.308,Z -93.945,A -90.000,B 90.000,C 0.000} C_DIS
LIN {X 105.397,Y -7.308,Z -94.122,A -90.000,B 90.000,C 0.000} C_DIS
LIN {X 105.507,Y -7.308,Z -94.522,A -90.000,B 90.000,C 0.000} C_DIS
LIN {X 105.517,Y -7.308,Z -94.560,A -90.000,B 90.000,C 0.000} C_DIS
LIN {X 105.585,Y -7.308,Z -94.815,A -90.000,B 90.000,C 0.000} C_DIS
LIN {X 105.594,Y -7.308,Z -94.851,A -90.000,B 90.000,C 0.000} C_DIS
LIN {X 105.641,Y -7.308,Z -95.027,A -90.000,B 90.000,C 0.000} C_DIS
LIN {X 105.737,Y -7.308,Z -95.437,A -90.000,B 90.000,C 0.000} C_DIS
LIN {X 105.913,Y -7.308,Z -96.162,A -90.000,B 90.000,C 0.000} C_DIS
LIN {X 106.117,Y -7.308,Z -97.033,A -90.000,B 90.000,C 0.000} C_DIS
LIN {X 106.202,Y -7.308,Z -97.402,A -90.000,B 90.000,C 0.000} C_DIS
LIN {X 106.440,Y -7.308,Z -98.459,A -90.000,B 90.000,C 0.000} C_DIS
LIN {X 106.517,Y -7.308,Z -98.798,A -90.000,B 90.000,C 0.000} C_DIS
LIN {X 106.800,Y -7.308,Z -100.095,A -90.000,B 90.000,C 0.000} C_DIS
LIN {X 106.868,Y -7.308,Z -100.399,A -90.000,B 90.000,C 0.000} C_DIS
LIN {X 106.881,Y -7.308,Z -100.460,A -90.000,B 90.000,C 0.000} C_DIS
LIN {X 106.883,Y -7.308,Z -100.472,A -90.000,B 90.000,C 0.000} C_DIS
LIN {X 107.164,Y -7.308,Z -101.791,A -90.000,B 90.000,C 0.000} C_DIS
LIN {X 107.234,Y -7.308,Z -102.110,A -90.000,B 90.000,C 0.000} C_DIS
LIN {X 107.238,Y -7.308,Z -102.130,A -90.000,B 90.000,C 0.000} C_DIS
LIN {X 107.270,Y -7.308,Z -102.275,A -90.000,B 90.000,C 0.000} C_DIS
LIN {X 107.460,Y -7.308,Z -103.141,A -90.000,B 90.000,C 0.000} C_DIS
LIN {X 107.733,Y -7.308,Z -104.447,A -90.000,B 90.000,C 0.000} C_DIS
LIN {X 107.928,Y -7.308,Z -105.372,A -90.000,B 90.000,C 0.000} C_DIS
LIN {X 108.229,Y -7.308,Z -106.872,A -90.000,B 90.000,C 0.000} C_DIS
LIN {X 108.422,Y -7.308,Z -107.844,A -90.000,B 90.000,C 0.000} C_DIS
LIN {X 108.734,Y -7.308,Z -109.493,A -90.000,B 90.000,C 0.000} C_DIS
LIN {X 108.913,Y -7.308,Z -110.487,A -90.000,B 90.000,C 0.000} C_DIS
LIN {X 109.220,Y -7.308,Z -112.253,A -90.000,B 90.000,C 0.000} C_DIS
LIN {X 109.269,Y -7.308,Z -112.560,A -90.000,B 90.000,C 0.000} C_DIS
LIN {X 109.295,Y -7.308,Z -112.723,A -90.000,B 90.000,C 0.000} C_DIS
LIN {X 109.589,Y -7.308,Z -114.634,A -90.000,B 90.000,C 0.000} C_DIS
LIN {X 109.736,Y -7.308,Z -115.563,A -90.000,B 90.000,C 0.000} C_DIS
LIN {X 110.013,Y -7.308,Z -117.591,A -90.000,B 90.000,C 0.000} C_DIS
LIN {X 110.129,Y -7.308,Z -118.425,A -90.000,B 90.000,C 0.000} C_DIS
LIN {X 110.386,Y -7.308,Z -120.558,A -90.000,B 90.000,C 0.000} C_DIS
LIN {X 110.472,Y -7.308,Z -121.255,A -90.000,B 90.000,C 0.000} C_DIS
LIN {X 110.704,Y -7.308,Z -123.464,A -90.000,B 90.000,C 0.000} C_DIS
LIN {X 110.763,Y -7.308,Z -123.999,A -90.000,B 90.000,C 0.000} C_DIS
LIN {X 110.962,Y -7.308,Z -126.234,A -90.000,B 90.000,C 0.000} C_DIS
LIN {X 110.997,Y -7.308,Z -126.603,A -90.000,B 90.000,C 0.000} C_DIS
LIN {X 111.160,Y -7.308,Z -128.944,A -90.000,B 90.000,C 0.000} C_DIS
LIN {X 111.178,Y -7.308,Z -129.172,A -90.000,B 90.000,C 0.000} C_DIS
LIN {X 111.201,Y -7.308,Z -129.607,A -90.000,B 90.000,C 0.000} C_DIS
LIN {X 111.202,Y -7.308,Z -129.640,A -90.000,B 90.000,C 0.000} C_DIS
LIN {X 111.203,Y -7.308,Z -129.647,A -90.000,B 90.000,C 0.000} C_DIS
LIN {X 111.288,Y -7.308,Z -131.428,A -90.000,B 90.000,C 0.000} C_DIS
LIN {X 111.296,Y -7.308,Z -131.583,A -90.000,B 90.000,C 0.000} C_DIS
LIN {X 111.305,Y -7.308,Z -131.736,A -90.000,B 90.000,C 0.000} C_DIS
LIN {X 111.312,Y -7.308,Z -131.867,A -90.000,B 90.000,C 0.000} C_DIS
LIN {X 111.329,Y -7.308,Z -132.186,A -90.000,B 90.000,C 0.000} C_DIS
LIN {X 111.337,Y -7.308,Z -132.333,A -90.000,B 90.000,C 0.000} C_DIS
LIN {X 111.390,Y -7.308,Z -134.348,A -90.000,B 90.000,C 0.000} C_DIS
LIN {X 111.416,Y -7.308,Z -135.135,A -90.000,B 90.000,C 0.000} C_DIS
LIN {X 111.426,Y -7.308,Z -135.907,A -90.000,B 90.000,C 0.000} C_DIS
LIN {X 111.444,Y -7.308,Z -138.207,A -90.000,B 90.000,C 0.000} C_DIS
LIN {X 111.441,Y -7.308,Z -138.887,A -90.000,B 90.000,C 0.000} C_DIS
LIN {X 111.418,Y -7.308,Z -141.511,A -90.000,B 90.000,C 0.000} C_DIS
LIN {X 111.408,Y -7.308,Z -142.082,A -90.000,B 90.000,C 0.000} C_DIS
LIN {X 111.339,Y -7.308,Z -145.011,A -90.000,B 90.000,C 0.000} C_DIS
LIN {X 111.324,Y -7.308,Z -145.462,A -90.000,B 90.000,C 0.000} C_DIS
LIN {X 111.203,Y -7.308,Z -148.668,A -90.000,B 90.000,C 0.000} C_DIS
LIN {X 111.191,Y -7.308,Z -148.973,A -90.000,B 90.000,C 0.000} C_DIS
LIN {X 111.190,Y -7.308,Z -149.004,A -90.000,B 90.000,C 0.000} C_DIS
LIN {X 111.175,Y -7.308,Z -149.328,A -90.000,B 90.000,C 0.000} C_DIS
LIN {X 110.995,Y -7.308,Z -152.779,A -90.000,B 90.000,C 0.000} C_DIS
LIN {X 110.984,Y -7.308,Z -152.975,A -90.000,B 90.000,C 0.000} C_DIS
LIN {X 110.751,Y -7.308,Z -156.635,A -90.000,B 90.000,C 0.000} C_DIS
LIN {X 110.746,Y -7.308,Z -156.705,A -90.000,B 90.000,C 0.000} C_DIS
LIN {X 110.579,Y -7.308,Z -158.991,A -90.000,B 90.000,C 0.000} C_DIS
LIN {X 110.479,Y -7.308,Z -160.358,A -90.000,B 90.000,C 0.000} C_DIS
LIN {X 110.468,Y -7.308,Z -160.520,A -90.000,B 90.000,C 0.000} C_DIS
LIN {X 110.425,Y -7.308,Z -161.093,A -90.000,B 90.000,C 0.000} C_DIS
LIN {X 110.414,Y -7.308,Z -161.239,A -90.000,B 90.000,C 0.000} C_DIS
LIN {X 110.178,Y -7.308,Z -164.191,A -90.000,B 90.000,C 0.000} C_DIS
LIN {X 110.149,Y -7.308,Z -164.544,A -90.000,B 90.000,C 0.000} C_DIS
LIN {X 110.141,Y -7.308,Z -164.645,A -90.000,B 90.000,C 0.000} C_DIS
LIN {X 109.901,Y -7.308,Z -167.454,A -90.000,B 90.000,C 0.000} C_DIS
LIN {X 109.854,Y -7.308,Z -168.058,A -90.000,B 90.000,C 0.000} C_DIS
LIN {X 109.825,Y -7.308,Z -168.421,A -90.000,B 90.000,C 0.000} C_DIS
LIN {X 109.817,Y -7.308,Z -168.512,A -90.000,B 90.000,C 0.000} C_DIS
LIN {X 109.539,Y -7.308,Z -171.553,A -90.000,B 90.000,C 0.000} C_DIS
LIN {X 109.480,Y -7.308,Z -172.271,A -90.000,B 90.000,C 0.000} C_DIS
LIN {X 109.190,Y -7.308,Z -175.204,A -90.000,B 90.000,C 0.000} C_DIS
LIN {X 109.132,Y -7.308,Z -175.846,A -90.000,B 90.000,C 0.000} C_DIS
LIN {X 108.837,Y -7.308,Z -178.588,A -90.000,B 90.000,C 0.000} C_DIS
LIN {X 108.780,Y -7.308,Z -179.161,A -90.000,B 90.000,C 0.000} C_DIS
LIN {X 108.724,Y -7.308,Z -179.674,A -90.000,B 90.000,C 0.000} C_DIS
LIN {X 108.428,Y -7.308,Z -182.143,A -90.000,B 90.000,C 0.000} C_DIS
LIN {X 108.371,Y -7.308,Z -182.609,A -90.000,B 90.000,C 0.000} C_DIS
LIN {X 108.076,Y -7.308,Z -184.865,A -90.000,B 90.000,C 0.000} C_DIS
LIN {X 108.018,Y -7.308,Z -185.302,A -90.000,B 90.000,C 0.000} C_DIS
LIN {X 107.951,Y -7.308,Z -185.795,A -90.000,B 90.000,C 0.000} C_DIS
LIN {X 107.917,Y -7.308,Z -186.050,A -90.000,B 90.000,C 0.000} C_DIS
LIN {X 107.712,Y -7.308,Z -187.505,A -90.000,B 90.000,C 0.000} C_DIS
LIN {X 107.569,Y -7.308,Z -188.533,A -90.000,B 90.000,C 0.000} C_DIS
LIN {X 107.363,Y -7.308,Z -189.927,A -90.000,B 90.000,C 0.000} C_DIS
LIN {X 107.220,Y -7.308,Z -190.924,A -90.000,B 90.000,C 0.000} C_DIS
LIN {X 107.011,Y -7.308,Z -192.314,A -90.000,B 90.000,C 0.000} C_DIS
LIN {X 106.855,Y -7.308,Z -193.353,A -90.000,B 90.000,C 0.000} C_DIS
LIN {X 106.615,Y -7.308,Z -194.889,A -90.000,B 90.000,C 0.000} C_DIS
LIN {X 106.436,Y -7.308,Z -196.028,A -90.000,B 90.000,C 0.000} C_DIS
LIN {X 106.135,Y -7.308,Z -197.874,A -90.000,B 90.000,C 0.000} C_DIS
LIN {X 105.927,Y -7.308,Z -199.146,A -90.000,B 90.000,C 0.000} C_DIS
LIN {X 105.531,Y -7.308,Z -201.493,A -90.000,B 90.000,C 0.000} C_DIS
LIN {X 105.294,Y -7.308,Z -202.891,A -90.000,B 90.000,C 0.000} C_DIS
LIN {X 104.761,Y -7.308,Z -205.966,A -90.000,B 90.000,C 0.000} C_DIS
LIN {X 104.513,Y -7.308,Z -207.319,A -90.000,B 90.000,C 0.000} C_DIS
LIN {X 103.817,Y -7.308,Z -211.065,A -90.000,B 90.000,C 0.000} C_DIS
LIN {X 103.577,Y -7.308,Z -212.239,A -90.000,B 90.000,C 0.000} C_DIS
LIN {X 102.691,Y -7.308,Z -216.562,A -90.000,B 90.000,C 0.000} C_DIS
LIN {X 102.612,Y -7.308,Z -216.920,A -90.000,B 90.000,C 0.000} C_DIS
LIN {X 102.596,Y -7.308,Z -216.993,A -90.000,B 90.000,C 0.000} C_DIS
LIN {X 102.382,Y -7.308,Z -217.907,A -90.000,B 90.000,C 0.000} C_DIS
LIN {X 101.282,Y -7.308,Z -222.664,A -90.000,B 90.000,C 0.000} C_DIS
LIN {X 99.890,Y -7.308,Z -227.862,A -90.000,B 90.000,C 0.000} C_DIS
LIN {X 99.773,Y -7.308,Z -228.285,A -90.000,B 90.000,C 0.000} C_DIS
LIN {X 98.104,Y -7.308,Z -233.819,A -90.000,B 90.000,C 0.000} C_DIS
LIN {X 98.052,Y -7.308,Z -233.986,A -90.000,B 90.000,C 0.000} C_DIS
LIN {X 97.018,Y -7.308,Z -237.114,A -90.000,B 90.000,C 0.000} C_DIS
LIN {X 96.258,Y -7.308,Z -239.395,A -90.000,B 90.000,C 0.000} C_DIS
LIN {X 96.094,Y -7.308,Z -239.886,A -90.000,B 90.000,C 0.000} C_DIS
LIN {X 96.081,Y -7.308,Z -239.927,A -90.000,B 90.000,C 0.000} C_DIS
LIN {X 95.952,Y -7.308,Z -240.302,A -90.000,B 90.000,C 0.000} C_DIS
LIN {X 95.884,Y -7.308,Z -240.498,A -90.000,B 90.000,C 0.000} C_DIS
LIN {X 94.791,Y -7.308,Z -243.561,A -90.000,B 90.000,C 0.000} C_DIS
LIN {X 94.791,Y -60.000,Z -243.561,A -90.000,B 90.000,C 0.000} C_DIS
LIN {X -120.015,Y -60.000,Z -237.460,A -90.000,B 90.000,C 0.000} C_DIS
LIN {X -120.015,Y -5.308,Z -237.460,A -90.000,B 90.000,C 0.000} C_DIS
LIN {X -119.172,Y -5.308,Z -236.901,A -90.000,B 90.000,C 0.000} C_DIS
LIN {X -113.005,Y -5.308,Z -232.837,A -90.000,B 90.000,C 0.000} C_DIS
LIN {X -111.728,Y -5.308,Z -231.997,A -90.000,B 90.000,C 0.000} C_DIS
LIN {X -111.669,Y -5.308,Z -231.958,A -90.000,B 90.000,C 0.000} C_DIS
LIN {X -111.330,Y -5.308,Z -231.736,A -90.000,B 90.000,C 0.000} C_DIS
LIN {X -103.939,Y -5.308,Z -226.926,A -90.000,B 90.000,C 0.000} C_DIS
LIN {X -103.598,Y -5.308,Z -226.705,A -90.000,B 90.000,C 0.000} C_DIS
LIN {X -101.055,Y -5.308,Z -225.084,A -90.000,B 90.000,C 0.000} C_DIS
LIN {X -95.690,Y -5.308,Z -221.679,A -90.000,B 90.000,C 0.000} C_DIS
LIN {X -95.537,Y -5.308,Z -221.585,A -90.000,B 90.000,C 0.000} C_DIS
LIN {X -87.566,Y -5.308,Z -216.674,A -90.000,B 90.000,C 0.000} C_DIS
LIN {X -87.179,Y -5.308,Z -216.437,A -90.000,B 90.000,C 0.000} C_DIS
LIN {X -79.939,Y -5.308,Z -212.156,A -90.000,B 90.000,C 0.000} C_DIS
LIN {X -78.634,Y -5.308,Z -211.389,A -90.000,B 90.000,C 0.000} C_DIS
LIN {X -72.736,Y -5.308,Z -207.978,A -90.000,B 90.000,C 0.000} C_DIS
LIN {X -70.208,Y -5.308,Z -206.528,A -90.000,B 90.000,C 0.000} C_DIS
LIN {X -65.747,Y -5.308,Z -203.965,A -90.000,B 90.000,C 0.000} C_DIS
LIN {X -62.281,Y -5.308,Z -201.994,A -90.000,B 90.000,C 0.000} C_DIS
LIN {X -59.150,Y -5.308,Z -200.172,A -90.000,B 90.000,C 0.000} C_DIS
LIN {X -55.235,Y -5.308,Z -197.917,A -90.000,B 90.000,C 0.000} C_DIS
LIN {X -53.281,Y -5.308,Z -196.731,A -90.000,B 90.000,C 0.000} C_DIS
LIN {X -53.187,Y -5.308,Z -196.674,A -90.000,B 90.000,C 0.000} C_DIS
LIN {X -52.895,Y -5.308,Z -196.498,A -90.000,B 90.000,C 0.000} C_DIS
LIN {X -49.799,Y -5.308,Z -194.634,A -90.000,B 90.000,C 0.000} C_DIS
LIN {X -48.060,Y -5.308,Z -193.524,A -90.000,B 90.000,C 0.000} C_DIS
LIN {X -47.534,Y -5.308,Z -193.189,A -90.000,B 90.000,C 0.000} C_DIS
LIN {X -45.047,Y -5.308,Z -191.611,A -90.000,B 90.000,C 0.000} C_DIS
LIN {X -43.247,Y -5.308,Z -190.399,A -90.000,B 90.000,C 0.000} C_DIS
LIN {X -41.052,Y -5.308,Z -188.928,A -90.000,B 90.000,C 0.000} C_DIS
LIN {X -39.506,Y -5.308,Z -187.834,A -90.000,B 90.000,C 0.000} C_DIS
LIN {X -37.571,Y -5.308,Z -186.471,A -90.000,B 90.000,C 0.000} C_DIS
LIN {X -35.936,Y -5.308,Z -185.279,A -90.000,B 90.000,C 0.000} C_DIS
LIN {X -35.806,Y -5.308,Z -185.185,A -90.000,B 90.000,C 0.000} C_DIS
LIN {X -34.615,Y -5.308,Z -184.314,A -90.000,B 90.000,C 0.000} C_DIS
LIN {X -34.610,Y -5.308,Z -184.310,A -90.000,B 90.000,C 0.000} C_DIS
LIN {X -34.599,Y -5.308,Z -184.302,A -90.000,B 90.000,C 0.000} C_DIS
LIN {X -33.164,Y -5.308,Z -183.208,A -90.000,B 90.000,C 0.000} C_DIS
LIN {X -33.110,Y -5.308,Z -183.166,A -90.000,B 90.000,C 0.000} C_DIS
LIN {X -31.791,Y -5.308,Z -182.156,A -90.000,B 90.000,C 0.000} C_DIS
LIN {X -30.417,Y -5.308,Z -181.042,A -90.000,B 90.000,C 0.000} C_DIS
LIN {X -29.126,Y -5.308,Z -179.992,A -90.000,B 90.000,C 0.000} C_DIS
LIN {X -28.065,Y -5.308,Z -179.060,A -90.000,B 90.000,C 0.000} C_DIS
LIN {X -27.955,Y -5.308,Z -178.963,A -90.000,B 90.000,C 0.000} C_DIS
LIN {X -26.986,Y -5.308,Z -178.110,A -90.000,B 90.000,C 0.000} C_DIS
LIN {X -26.065,Y -5.308,Z -177.212,A -90.000,B 90.000,C 0.000} C_DIS
LIN {X -26.023,Y -5.308,Z -177.170,A -90.000,B 90.000,C 0.000} C_DIS
LIN {X -25.960,Y -5.308,Z -177.110,A -90.000,B 90.000,C 0.000} C_DIS
LIN {X -25.051,Y -5.308,Z -176.222,A -90.000,B 90.000,C 0.000} C_DIS
LIN {X -24.214,Y -5.308,Z -175.296,A -90.000,B 90.000,C 0.000} C_DIS
LIN {X -24.212,Y -5.308,Z -175.293,A -90.000,B 90.000,C 0.000} C_DIS
LIN {X -24.054,Y -5.308,Z -175.119,A -90.000,B 90.000,C 0.000} C_DIS
LIN {X -23.546,Y -5.308,Z -174.553,A -90.000,B 90.000,C 0.000} C_DIS
LIN {X -23.546,Y -5.308,Z -174.552,A -90.000,B 90.000,C 0.000} C_DIS
LIN {X -22.720,Y -5.308,Z -173.495,A -90.000,B 90.000,C 0.000} C_DIS
LIN {X -22.716,Y -5.308,Z -173.490,A -90.000,B 90.000,C 0.000} C_DIS
LIN {X -22.638,Y -5.308,Z -173.389,A -90.000,B 90.000,C 0.000} C_DIS
LIN {X -22.633,Y -5.308,Z -173.383,A -90.000,B 90.000,C 0.000} C_DIS
LIN {X -22.120,Y -5.308,Z -172.717,A -90.000,B 90.000,C 0.000} C_DIS
LIN {X -22.115,Y -5.308,Z -172.711,A -90.000,B 90.000,C 0.000} C_DIS
LIN {X -21.349,Y -5.308,Z -171.562,A -90.000,B 90.000,C 0.000} C_DIS
LIN {X -21.309,Y -5.308,Z -171.501,A -90.000,B 90.000,C 0.000} C_DIS
LIN {X -20.850,Y -5.308,Z -170.801,A -90.000,B 90.000,C 0.000} C_DIS
LIN {X -20.849,Y -5.308,Z -170.801,A -90.000,B 90.000,C 0.000} C_DIS
LIN {X -20.846,Y -5.308,Z -170.795,A -90.000,B 90.000,C 0.000} C_DIS
LIN {X -20.227,Y -5.308,Z -169.709,A -90.000,B 90.000,C 0.000} C_DIS
LIN {X -20.223,Y -5.308,Z -169.703,A -90.000,B 90.000,C 0.000} C_DIS
LIN {X -19.699,Y -5.308,Z -168.770,A -90.000,B 90.000,C 0.000} C_DIS
LIN {X -19.692,Y -5.308,Z -168.755,A -90.000,B 90.000,C 0.000} C_DIS
LIN {X -19.122,Y -5.308,Z -167.591,A -90.000,B 90.000,C 0.000} C_DIS
LIN {X -19.113,Y -5.308,Z -167.571,A -90.000,B 90.000,C 0.000} C_DIS
LIN {X -19.099,Y -5.308,Z -167.542,A -90.000,B 90.000,C 0.000} C_DIS
LIN {X -19.095,Y -5.308,Z -167.534,A -90.000,B 90.000,C 0.000} C_DIS
LIN {X -18.593,Y -5.308,Z -166.497,A -90.000,B 90.000,C 0.000} C_DIS
LIN {X -18.592,Y -5.308,Z -166.496,A -90.000,B 90.000,C 0.000} C_DIS
LIN {X -18.182,Y -5.308,Z -165.489,A -90.000,B 90.000,C 0.000} C_DIS
LIN {X -18.121,Y -5.308,Z -165.340,A -90.000,B 90.000,C 0.000} C_DIS
LIN {X -17.800,Y -5.308,Z -164.549,A -90.000,B 90.000,C 0.000} C_DIS
LIN {X -17.505,Y -5.308,Z -163.586,A -90.000,B 90.000,C 0.000} C_DIS
LIN {X -17.503,Y -5.308,Z -163.582,A -90.000,B 90.000,C 0.000} C_DIS
LIN {X -17.391,Y -5.308,Z -163.214,A -90.000,B 90.000,C 0.000} C_DIS
LIN {X -17.337,Y -5.308,Z -163.043,A -90.000,B 90.000,C 0.000} C_DIS
LIN {X -17.228,Y -5.308,Z -162.316,A -90.000,B 90.000,C 0.000} C_DIS
LIN {X -17.218,Y -5.308,Z -162.258,A -90.000,B 90.000,C 0.000} C_DIS
LIN {X -17.218,Y -5.308,Z -162.257,A -90.000,B 90.000,C 0.000} C_DIS
LIN {X -17.197,Y -5.308,Z -162.129,A -90.000,B 90.000,C 0.000} C_DIS
LIN {X -17.211,Y -5.308,Z -161.822,A -90.000,B 90.000,C 0.000} C_DIS
LIN {X -17.213,Y -5.308,Z -161.726,A -90.000,B 90.000,C 0.000} C_DIS
LIN {X -17.215,Y -5.308,Z -161.670,A -90.000,B 90.000,C 0.000} C_DIS
LIN {X -17.249,Y -5.308,Z -161.532,A -90.000,B 90.000,C 0.000} C_DIS
LIN {X -17.269,Y -5.308,Z -161.444,A -90.000,B 90.000,C 0.000} C_DIS
LIN {X -17.314,Y -5.308,Z -161.243,A -90.000,B 90.000,C 0.000} C_DIS
LIN {X -17.321,Y -5.308,Z -161.226,A -90.000,B 90.000,C 0.000} C_DIS
LIN {X -17.411,Y -5.308,Z -160.999,A -90.000,B 90.000,C 0.000} C_DIS
LIN {X -17.480,Y -5.308,Z -160.827,A -90.000,B 90.000,C 0.000} C_DIS
LIN {X -17.638,Y -5.308,Z -160.396,A -90.000,B 90.000,C 0.000} C_DIS
LIN {X -17.880,Y -5.308,Z -159.852,A -90.000,B 90.000,C 0.000} C_DIS
LIN {X -17.989,Y -5.308,Z -159.610,A -90.000,B 90.000,C 0.000} C_DIS
LIN {X -18.058,Y -5.308,Z -159.441,A -90.000,B 90.000,C 0.000} C_DIS
LIN {X -18.387,Y -5.308,Z -158.857,A -90.000,B 90.000,C 0.000} C_DIS
LIN {X -18.393,Y -5.308,Z -158.848,A -90.000,B 90.000,C 0.000} C_DIS
LIN {X -18.500,Y -5.308,Z -158.659,A -90.000,B 90.000,C 0.000} C_DIS
LIN {X -18.504,Y -5.308,Z -158.650,A -90.000,B 90.000,C 0.000} C_DIS
LIN {X -18.506,Y -5.308,Z -158.647,A -90.000,B 90.000,C 0.000} C_DIS
LIN {X -18.636,Y -5.308,Z -158.401,A -90.000,B 90.000,C 0.000} C_DIS
LIN {X -18.755,Y -5.308,Z -158.233,A -90.000,B 90.000,C 0.000} C_DIS
LIN {X -18.963,Y -5.308,Z -157.938,A -90.000,B 90.000,C 0.000} C_DIS
LIN {X -19.358,Y -5.308,Z -157.379,A -90.000,B 90.000,C 0.000} C_DIS
LIN {X -19.370,Y -5.308,Z -157.362,A -90.000,B 90.000,C 0.000} C_DIS
LIN {X -19.588,Y -5.308,Z -157.049,A -90.000,B 90.000,C 0.000} C_DIS
LIN {X -19.605,Y -5.308,Z -157.028,A -90.000,B 90.000,C 0.000} C_DIS
LIN {X -19.868,Y -5.308,Z -156.715,A -90.000,B 90.000,C 0.000} C_DIS
LIN {X -19.870,Y -5.308,Z -156.713,A -90.000,B 90.000,C 0.000} C_DIS
LIN {X -20.307,Y -5.308,Z -156.192,A -90.000,B 90.000,C 0.000} C_DIS
LIN {X -21.079,Y -5.308,Z -155.273,A -90.000,B 90.000,C 0.000} C_DIS
LIN {X -21.081,Y -5.308,Z -155.270,A -90.000,B 90.000,C 0.000} C_DIS
LIN {X -21.082,Y -5.308,Z -155.270,A -90.000,B 90.000,C 0.000} C_DIS
LIN {X -21.150,Y -5.308,Z -155.186,A -90.000,B 90.000,C 0.000} C_DIS
LIN {X -23.178,Y -5.308,Z -153.058,A -90.000,B 90.000,C 0.000} C_DIS
LIN {X -23.198,Y -5.308,Z -153.037,A -90.000,B 90.000,C 0.000} C_DIS
LIN {X -23.557,Y -5.308,Z -152.652,A -90.000,B 90.000,C 0.000} C_DIS
LIN {X -26.064,Y -5.308,Z -150.025,A -90.000,B 90.000,C 0.000} C_DIS
LIN {X -26.524,Y -5.308,Z -149.535,A -90.000,B 90.000,C 0.000} C_DIS
LIN {X -29.152,Y -5.308,Z -146.575,A -90.000,B 90.000,C 0.000} C_DIS
LIN {X -29.638,Y -5.308,Z -146.019,A -90.000,B 90.000,C 0.000} C_DIS
LIN {X -29.906,Y -5.308,Z -145.708,A -90.000,B 90.000,C 0.000} C_DIS
LIN {X -29.956,Y -5.308,Z -145.650,A -90.000,B 90.000,C 0.000} C_DIS
LIN {X -32.493,Y -5.308,Z -142.362,A -90.000,B 90.000,C 0.000} C_DIS
LIN {X -32.928,Y -5.308,Z -141.790,A -90.000,B 90.000,C 0.000} C_DIS
LIN {X -33.165,Y -5.308,Z -141.449,A -90.000,B 90.000,C 0.000} C_DIS
LIN {X -33.206,Y -5.308,Z -141.391,A -90.000,B 90.000,C 0.000} C_DIS
LIN {X -35.450,Y -5.308,Z -137.735,A -90.000,B 90.000,C 0.000} C_DIS
LIN {X -35.746,Y -5.308,Z -137.245,A -90.000,B 90.000,C 0.000} C_DIS
LIN {X -35.760,Y -5.308,Z -137.222,A -90.000,B 90.000,C 0.000} C_DIS
LIN {X -35.847,Y -5.308,Z -137.064,A -90.000,B 90.000,C 0.000} C_DIS
LIN {X -35.961,Y -5.308,Z -136.857,A -90.000,B 90.000,C 0.000} C_DIS
LIN {X -35.982,Y -5.308,Z -136.819,A -90.000,B 90.000,C 0.000} C_DIS
LIN {X -37.196,Y -5.308,Z -134.467,A -90.000,B 90.000,C 0.000} C_DIS
LIN {X -37.196,Y -60.000,Z -134.467,A -90.000,B 90.000,C 0.000} C_DIS
LIN {X -42.720,Y -60.000,Z -122.406,A -90.000,B 90.000,C 0.000} C_DIS
LIN {X -42.720,Y -5.308,Z -122.406,A -90.000,B 90.000,C 0.000} C_DIS
LIN {X -43.112,Y -5.308,Z -121.622,A -90.000,B 90.000,C 0.000} C_DIS
LIN {X -43.116,Y -5.308,Z -121.614,A -90.000,B 90.000,C 0.000} C_DIS
LIN {X -43.222,Y -5.308,Z -121.437,A -90.000,B 90.000,C 0.000} C_DIS
LIN {X -43.224,Y -5.308,Z -121.434,A -90.000,B 90.000,C 0.000} C_DIS
LIN {X -43.720,Y -5.308,Z -120.605,A -90.000,B 90.000,C 0.000} C_DIS
LIN {X -43.874,Y -5.308,Z -120.347,A -90.000,B 90.000,C 0.000} C_DIS
LIN {X -44.040,Y -5.308,Z -120.112,A -90.000,B 90.000,C 0.000} C_DIS
LIN {X -44.042,Y -5.308,Z -120.109,A -90.000,B 90.000,C 0.000} C_DIS
LIN {X -44.741,Y -5.308,Z -119.117,A -90.000,B 90.000,C 0.000} C_DIS
LIN {X -45.920,Y -5.308,Z -117.583,A -90.000,B 90.000,C 0.000} C_DIS
LIN {X -46.250,Y -5.308,Z -117.158,A -90.000,B 90.000,C 0.000} C_DIS
LIN {X -47.641,Y -5.308,Z -115.415,A -90.000,B 90.000,C 0.000} C_DIS
LIN {X -48.072,Y -5.308,Z -114.880,A -90.000,B 90.000,C 0.000} C_DIS
LIN {X -49.602,Y -5.308,Z -112.986,A -90.000,B 90.000,C 0.000} C_DIS
LIN {X -50.138,Y -5.308,Z -112.326,A -90.000,B 90.000,C 0.000} C_DIS
LIN {X -51.714,Y -5.308,Z -110.365,A -90.000,B 90.000,C 0.000} C_DIS
LIN {X -52.380,Y -5.308,Z -109.534,A -90.000,B 90.000,C 0.000} C_DIS
LIN {X -53.233,Y -5.308,Z -108.433,A -90.000,B 90.000,C 0.000} C_DIS
LIN {X -54.725,Y -5.308,Z -106.541,A -90.000,B 90.000,C 0.000} C_DIS
LIN {X -55.843,Y -5.308,Z -105.100,A -90.000,B 90.000,C 0.000} C_DIS
LIN {X -57.129,Y -5.308,Z -103.485,A -90.000,B 90.000,C 0.000} C_DIS
LIN {X -57.417,Y -5.308,Z -103.126,A -90.000,B 90.000,C 0.000} C_DIS
LIN {X -57.546,Y -5.308,Z -102.964,A -90.000,B 90.000,C 0.000} C_DIS
LIN {X -58.433,Y -5.308,Z -101.860,A -90.000,B 90.000,C 0.000} C_DIS
LIN {X -58.448,Y -5.308,Z -101.841,A -90.000,B 90.000,C 0.000} C_DIS
LIN {X -59.381,Y -5.308,Z -100.711,A -90.000,B 90.000,C 0.000} C_DIS
LIN {X -60.260,Y -5.308,Z -99.693,A -90.000,B 90.000,C 0.000} C_DIS
LIN {X -60.290,Y -5.308,Z -99.658,A -90.000,B 90.000,C 0.000} C_DIS
LIN {X -61.556,Y -5.308,Z -98.229,A -90.000,B 90.000,C 0.000} C_DIS
LIN {X -61.564,Y -5.308,Z -98.221,A -90.000,B 90.000,C 0.000} C_DIS
LIN {X -62.665,Y -5.308,Z -97.121,A -90.000,B 90.000,C 0.000} C_DIS
LIN {X -63.131,Y -5.308,Z -96.644,A -90.000,B 90.000,C 0.000} C_DIS
LIN {X -63.794,Y -5.308,Z -95.966,A -90.000,B 90.000,C 0.000} C_DIS
LIN {X -63.795,Y -5.308,Z -95.965,A -90.000,B 90.000,C 0.000} C_DIS
LIN {X -65.080,Y -5.308,Z -94.824,A -90.000,B 90.000,C 0.000} C_DIS
LIN {X -65.263,Y -5.308,Z -94.661,A -90.000,B 90.000,C 0.000} C_DIS
LIN {X -65.814,Y -5.308,Z -94.165,A -90.000,B 90.000,C 0.000} C_DIS
LIN {X -65.822,Y -5.308,Z -94.157,A -90.000,B 90.000,C 0.000} C_DIS
LIN {X -65.865,Y -5.308,Z -94.119,A -90.000,B 90.000,C 0.000} C_DIS
LIN {X -67.212,Y -5.308,Z -93.048,A -90.000,B 90.000,C 0.000} C_DIS
LIN {X -67.466,Y -5.308,Z -92.845,A -90.000,B 90.000,C 0.000} C_DIS
LIN {X -67.798,Y -5.308,Z -92.580,A -90.000,B 90.000,C 0.000} C_DIS
LIN {X -69.403,Y -5.308,Z -91.420,A -90.000,B 90.000,C 0.000} C_DIS
LIN {X -69.412,Y -5.308,Z -91.413,A -90.000,B 90.000,C 0.000} C_DIS
LIN {X -70.020,Y -5.308,Z -90.973,A -90.000,B 90.000,C 0.000} C_DIS
LIN {X -70.568,Y -5.308,Z -90.602,A -90.000,B 90.000,C 0.000} C_DIS
LIN {X -72.257,Y -5.308,Z -89.469,A -90.000,B 90.000,C 0.000} C_DIS
LIN {X -72.496,Y -5.308,Z -89.314,A -90.000,B 90.000,C 0.000} C_DIS
LIN {X -72.512,Y -5.308,Z -89.304,A -90.000,B 90.000,C 0.000} C_DIS
LIN {X -73.212,Y -5.308,Z -88.857,A -90.000,B 90.000,C 0.000} C_DIS
LIN {X -73.463,Y -5.308,Z -88.697,A -90.000,B 90.000,C 0.000} C_DIS
LIN {X -73.738,Y -5.308,Z -88.522,A -90.000,B 90.000,C 0.000} C_DIS
LIN {X -74.102,Y -5.308,Z -88.288,A -90.000,B 90.000,C 0.000} C_DIS
LIN {X -74.151,Y -5.308,Z -88.256,A -90.000,B 90.000,C 0.000} C_DIS
LIN {X -74.576,Y -5.308,Z -87.990,A -90.000,B 90.000,C 0.000} C_DIS
LIN {X -75.478,Y -5.308,Z -87.423,A -90.000,B 90.000,C 0.000} C_DIS
LIN {X -76.026,Y -5.308,Z -87.082,A -90.000,B 90.000,C 0.000} C_DIS
LIN {X -76.962,Y -5.308,Z -86.487,A -90.000,B 90.000,C 0.000} C_DIS
LIN {X -77.843,Y -5.308,Z -85.929,A -90.000,B 90.000,C 0.000} C_DIS
LIN {X -78.000,Y -5.308,Z -85.830,A -90.000,B 90.000,C 0.000} C_DIS
LIN {X -78.245,Y -5.308,Z -85.674,A -90.000,B 90.000,C 0.000} C_DIS
LIN {X -78.745,Y -5.308,Z -85.337,A -90.000,B 90.000,C 0.000} C_DIS
LIN {X -79.805,Y -5.308,Z -84.616,A -90.000,B 90.000,C 0.000} C_DIS
LIN {X -80.031,Y -5.308,Z -84.454,A -90.000,B 90.000,C 0.000} C_DIS
LIN {X -81.158,Y -5.308,Z -83.634,A -90.000,B 90.000,C 0.000} C_DIS
LIN {X -81.226,Y -5.308,Z -83.583,A -90.000,B 90.000,C 0.000} C_DIS
LIN {X -82.073,Y -5.308,Z -82.933,A -90.000,B 90.000,C 0.000} C_DIS
LIN {X -82.368,Y -5.308,Z -82.706,A -90.000,B 90.000,C 0.000} C_DIS
LIN {X -82.608,Y -5.308,Z -82.515,A -90.000,B 90.000,C 0.000} C_DIS
LIN {X -82.643,Y -5.308,Z -82.488,A -90.000,B 90.000,C 0.000} C_DIS
LIN {X -82.725,Y -5.308,Z -82.423,A -90.000,B 90.000,C 0.000} C_DIS
LIN {X -82.778,Y -5.308,Z -82.380,A -90.000,B 90.000,C 0.000} C_DIS
LIN {X -83.805,Y -5.308,Z -81.564,A -90.000,B 90.000,C 0.000} C_DIS
LIN {X -83.910,Y -5.308,Z -81.480,A -90.000,B 90.000,C 0.000} C_DIS
LIN {X -83.983,Y -5.308,Z -81.422,A -90.000,B 90.000,C 0.000} C_DIS
LIN {X -84.359,Y -5.308,Z -81.122,A -90.000,B 90.000,C 0.000} C_DIS
LIN {X -84.549,Y -5.308,Z -80.970,A -90.000,B 90.000,C 0.000} C_DIS
LIN {X -84.829,Y -5.308,Z -80.747,A -90.000,B 90.000,C 0.000} C_DIS
LIN {X -84.867,Y -5.308,Z -80.717,A -90.000,B 90.000,C 0.000} C_DIS
LIN {X -85.390,Y -5.308,Z -80.300,A -90.000,B 90.000,C 0.000} C_DIS
LIN {X -85.481,Y -5.308,Z -80.232,A -90.000,B 90.000,C 0.000} C_DIS
LIN {X -85.539,Y -5.308,Z -80.187,A -90.000,B 90.000,C 0.000} C_DIS
LIN {X -86.308,Y -5.308,Z -79.583,A -90.000,B 90.000,C 0.000} C_DIS
LIN {X -86.412,Y -5.308,Z -79.506,A -90.000,B 90.000,C 0.000} C_DIS
LIN {X -86.437,Y -5.308,Z -79.487,A -90.000,B 90.000,C 0.000} C_DIS
LIN {X -86.445,Y -5.308,Z -79.481,A -90.000,B 90.000,C 0.000} C_DIS
LIN {X -87.008,Y -5.308,Z -79.051,A -90.000,B 90.000,C 0.000} C_DIS
LIN {X -87.131,Y -5.308,Z -78.961,A -90.000,B 90.000,C 0.000} C_DIS
LIN {X -87.173,Y -5.308,Z -78.931,A -90.000,B 90.000,C 0.000} C_DIS
LIN {X -87.290,Y -5.308,Z -78.846,A -90.000,B 90.000,C 0.000} C_DIS
LIN {X -87.682,Y -5.308,Z -78.559,A -90.000,B 90.000,C 0.000} C_DIS
LIN {X -87.695,Y -5.308,Z -78.549,A -90.000,B 90.000,C 0.000} C_DIS
LIN {X -88.082,Y -5.308,Z -78.269,A -90.000,B 90.000,C 0.000} C_DIS
LIN {X -88.091,Y -5.308,Z -78.262,A -90.000,B 90.000,C 0.000} C_DIS
LIN {X -88.199,Y -5.308,Z -78.188,A -90.000,B 90.000,C 0.000} C_DIS
LIN {X -88.485,Y -5.308,Z -77.991,A -90.000,B 90.000,C 0.000} C_DIS
LIN {X -88.620,Y -5.308,Z -77.895,A -90.000,B 90.000,C 0.000} C_DIS
LIN {X -88.632,Y -5.308,Z -77.888,A -90.000,B 90.000,C 0.000} C_DIS
LIN {X -88.646,Y -5.308,Z -77.879,A -90.000,B 90.000,C 0.000} C_DIS
LIN {X -88.822,Y -5.308,Z -77.767,A -90.000,B 90.000,C 0.000} C_DIS
LIN {X -89.145,Y -5.308,Z -77.554,A -90.000,B 90.000,C 0.000} C_DIS
LIN {X -89.156,Y -5.308,Z -77.546,A -90.000,B 90.000,C 0.000} C_DIS
LIN {X -89.157,Y -5.308,Z -77.545,A -90.000,B 90.000,C 0.000} C_DIS
LIN {X -89.199,Y -5.308,Z -77.522,A -90.000,B 90.000,C 0.000} C_DIS
LIN {X -89.228,Y -5.308,Z -77.506,A -90.000,B 90.000,C 0.000} C_DIS
LIN {X -89.477,Y -5.308,Z -77.365,A -90.000,B 90.000,C 0.000} C_DIS
LIN {X -89.481,Y -5.308,Z -77.362,A -90.000,B 90.000,C 0.000} C_DIS
LIN {X -89.485,Y -5.308,Z -77.360,A -90.000,B 90.000,C 0.000} C_DIS
LIN {X -89.632,Y -5.308,Z -77.272,A -90.000,B 90.000,C 0.000} C_DIS
LIN {X -89.650,Y -5.308,Z -77.263,A -90.000,B 90.000,C 0.000} C_DIS
LIN {X -89.677,Y -5.308,Z -77.249,A -90.000,B 90.000,C 0.000} C_DIS
LIN {X -89.714,Y -5.308,Z -77.230,A -90.000,B 90.000,C 0.000} C_DIS
LIN {X -89.743,Y -5.308,Z -77.216,A -90.000,B 90.000,C 0.000} C_DIS
LIN {X -89.901,Y -5.308,Z -77.135,A -90.000,B 90.000,C 0.000} C_DIS
LIN {X -89.944,Y -5.308,Z -77.118,A -90.000,B 90.000,C 0.000} C_DIS
LIN {X -89.948,Y -5.308,Z -77.117,A -90.000,B 90.000,C 0.000} C_DIS
LIN {X -89.951,Y -5.308,Z -77.115,A -90.000,B 90.000,C 0.000} C_DIS
LIN {X -89.984,Y -5.308,Z -77.102,A -90.000,B 90.000,C 0.000} C_DIS
LIN {X -90.016,Y -5.308,Z -77.094,A -90.000,B 90.000,C 0.000} C_DIS
LIN {X -90.036,Y -5.308,Z -77.089,A -90.000,B 90.000,C 0.000} C_DIS
LIN {X -90.041,Y -5.308,Z -77.088,A -90.000,B 90.000,C 0.000} C_DIS
LIN {X -90.048,Y -5.308,Z -77.086,A -90.000,B 90.000,C 0.000} C_DIS
LIN {X -90.084,Y -5.308,Z -77.082,A -90.000,B 90.000,C 0.000} C_DIS
LIN {X -90.098,Y -5.308,Z -77.081,A -90.000,B 90.000,C 0.000} C_DIS
LIN {X -90.148,Y -5.308,Z -77.075,A -90.000,B 90.000,C 0.000} C_DIS
LIN {X -90.203,Y -5.308,Z -77.069,A -90.000,B 90.000,C 0.000} C_DIS
LIN {X -90.367,Y -5.308,Z -77.067,A -90.000,B 90.000,C 0.000} C_DIS
LIN {X -90.536,Y -5.308,Z -77.064,A -90.000,B 90.000,C 0.000} C_DIS
LIN {X -90.588,Y -5.308,Z -77.064,A -90.000,B 90.000,C 0.000} C_DIS
LIN {X -90.713,Y -5.308,Z -77.065,A -90.000,B 90.000,C 0.000} C_DIS
LIN {X -90.760,Y -5.308,Z -77.066,A -90.000,B 90.000,C 0.000} C_DIS
LIN {X -90.948,Y -5.308,Z -77.073,A -90.000,B 90.000,C 0.000} C_DIS
LIN {X -90.976,Y -5.308,Z -77.075,A -90.000,B 90.000,C 0.000} C_DIS
LIN {X -91.207,Y -5.308,Z -77.092,A -90.000,B 90.000,C 0.000} C_DIS
LIN {X -91.385,Y -5.308,Z -77.101,A -90.000,B 90.000,C 0.000} C_DIS
LIN {X -91.468,Y -5.308,Z -77.105,A -90.000,B 90.000,C 0.000} C_DIS
LIN {X -91.472,Y -5.308,Z -77.105,A -90.000,B 90.000,C 0.000} C_DIS
LIN {X -92.065,Y -5.308,Z -77.156,A -90.000,B 90.000,C 0.000} C_DIS
LIN {X -92.212,Y -5.308,Z -77.168,A -90.000,B 90.000,C 0.000} C_DIS
LIN {X -92.274,Y -5.308,Z -77.172,A -90.000,B 90.000,C 0.000} C_DIS
LIN {X -92.677,Y -5.308,Z -77.192,A -90.000,B 90.000,C 0.000} C_DIS
LIN {X -92.880,Y -5.308,Z -77.201,A -90.000,B 90.000,C 0.000} C_DIS
LIN {X -93.483,Y -5.308,Z -77.218,A -90.000,B 90.000,C 0.000} C_DIS
LIN {X -93.699,Y -5.308,Z -77.229,A -90.000,B 90.000,C 0.000} C_DIS
LIN {X -93.817,Y -5.308,Z -77.235,A -90.000,B 90.000,C 0.000} C_DIS
LIN {X -94.542,Y -5.308,Z -77.216,A -90.000,B 90.000,C 0.000} C_DIS
LIN {X -95.044,Y -5.308,Z -77.220,A -90.000,B 90.000,C 0.000} C_DIS
LIN {X -95.284,Y -5.308,Z -77.206,A -90.000,B 90.000,C 0.000} C_DIS
LIN {X -95.510,Y -5.308,Z -77.193,A -90.000,B 90.000,C 0.000} C_DIS
LIN {X -95.725,Y -5.308,Z -77.168,A -90.000,B 90.000,C 0.000} C_DIS
LIN {X -95.869,Y -5.308,Z -77.152,A -90.000,B 90.000,C 0.000} C_DIS
LIN {X -96.043,Y -5.308,Z -77.131,A -90.000,B 90.000,C 0.000} C_DIS
LIN {X -96.764,Y -5.308,Z -77.070,A -90.000,B 90.000,C 0.000} C_DIS
LIN {X -96.765,Y -5.308,Z -77.070,A -90.000,B 90.000,C 0.000} C_DIS
LIN {X -96.844,Y -5.308,Z -77.062,A -90.000,B 90.000,C 0.000} C_DIS
LIN {X -97.009,Y -5.308,Z -77.035,A -90.000,B 90.000,C 0.000} C_DIS
LIN {X -97.305,Y -5.308,Z -76.986,A -90.000,B 90.000,C 0.000} C_DIS
LIN {X -97.480,Y -5.308,Z -76.944,A -90.000,B 90.000,C 0.000} C_DIS
LIN {X -97.527,Y -5.308,Z -76.933,A -90.000,B 90.000,C 0.000} C_DIS
LIN {X -97.597,Y -5.308,Z -76.918,A -90.000,B 90.000,C 0.000} C_DIS
LIN {X -98.686,Y -5.308,Z -76.687,A -90.000,B 90.000,C 0.000} C_DIS
LIN {X -99.029,Y -5.308,Z -76.593,A -90.000,B 90.000,C 0.000} C_DIS
LIN {X -99.128,Y -5.308,Z -76.566,A -90.000,B 90.000,C 0.000} C_DIS
LIN {X -99.194,Y -5.308,Z -76.544,A -90.000,B 90.000,C 0.000} C_DIS
LIN {X -99.311,Y -5.308,Z -76.498,A -90.000,B 90.000,C 0.000} C_DIS
LIN {X -99.480,Y -5.308,Z -76.437,A -90.000,B 90.000,C 0.000} C_DIS
LIN {X -99.667,Y -5.308,Z -76.368,A -90.000,B 90.000,C 0.000} C_DIS
LIN {X -100.678,Y -5.308,Z -75.998,A -90.000,B 90.000,C 0.000} C_DIS
LIN {X -100.996,Y -5.308,Z -75.872,A -90.000,B 90.000,C 0.000} C_DIS
LIN {X -101.105,Y -5.308,Z -75.829,A -90.000,B 90.000,C 0.000} C_DIS
LIN {X -101.163,Y -5.308,Z -75.800,A -90.000,B 90.000,C 0.000} C_DIS
LIN {X -101.269,Y -5.308,Z -75.744,A -90.000,B 90.000,C 0.000} C_DIS
LIN {X -101.576,Y -5.308,Z -75.582,A -90.000,B 90.000,C 0.000} C_DIS
LIN {X -101.789,Y -5.308,Z -75.462,A -90.000,B 90.000,C 0.000} C_DIS
LIN {X -101.848,Y -5.308,Z -75.430,A -90.000,B 90.000,C 0.000} C_DIS
LIN {X -103.128,Y -5.308,Z -74.731,A -90.000,B 90.000,C 0.000} C_DIS
LIN {X -103.195,Y -5.308,Z -74.690,A -90.000,B 90.000,C 0.000} C_DIS
LIN {X -103.321,Y -5.308,Z -74.605,A -90.000,B 90.000,C 0.000} C_DIS
LIN {X -103.582,Y -5.308,Z -74.429,A -90.000,B 90.000,C 0.000} C_DIS
LIN {X -103.874,Y -5.308,Z -74.223,A -90.000,B 90.000,C 0.000} C_DIS
LIN {X -104.009,Y -5.308,Z -74.129,A -90.000,B 90.000,C 0.000} C_DIS
LIN {X -104.059,Y -5.308,Z -74.094,A -90.000,B 90.000,C 0.000} C_DIS
LIN {X -105.119,Y -5.308,Z -73.363,A -90.000,B 90.000,C 0.000} C_DIS
LIN {X -105.126,Y -5.308,Z -73.358,A -90.000,B 90.000,C 0.000} C_DIS
LIN {X -105.136,Y -5.308,Z -73.351,A -90.000,B 90.000,C 0.000} C_DIS
LIN {X -105.188,Y -5.308,Z -73.314,A -90.000,B 90.000,C 0.000} C_DIS
LIN {X -105.390,Y -5.308,Z -73.146,A -90.000,B 90.000,C 0.000} C_DIS
LIN {X -105.471,Y -5.308,Z -73.079,A -90.000,B 90.000,C 0.000} C_DIS
LIN {X -105.815,Y -5.308,Z -72.794,A -90.000,B 90.000,C 0.000} C_DIS
LIN {X -106.597,Y -5.308,Z -72.155,A -90.000,B 90.000,C 0.000} C_DIS
LIN {X -106.604,Y -5.308,Z -72.149,A -90.000,B 90.000,C 0.000} C_DIS
LIN {X -106.646,Y -5.308,Z -72.115,A -90.000,B 90.000,C 0.000} C_DIS
LIN {X -106.813,Y -5.308,Z -71.974,A -90.000,B 90.000,C 0.000} C_DIS
LIN {X -107.047,Y -5.308,Z -71.776,A -90.000,B 90.000,C 0.000} C_DIS
LIN {X -107.188,Y -5.308,Z -71.640,A -90.000,B 90.000,C 0.000} C_DIS
LIN {X -107.255,Y -5.308,Z -71.576,A -90.000,B 90.000,C 0.000} C_DIS
LIN {X -107.957,Y -5.308,Z -70.900,A -90.000,B 90.000,C 0.000} C_DIS
LIN {X -108.285,Y -5.308,Z -70.589,A -90.000,B 90.000,C 0.000} C_DIS
LIN {X -108.289,Y -5.308,Z -70.585,A -90.000,B 90.000,C 0.000} C_DIS
LIN {X -108.325,Y -5.308,Z -70.551,A -90.000,B 90.000,C 0.000} C_DIS
LIN {X -108.352,Y -5.308,Z -70.524,A -90.000,B 90.000,C 0.000} C_DIS
LIN {X -108.363,Y -5.308,Z -70.513,A -90.000,B 90.000,C 0.000} C_DIS
LIN {X -108.629,Y -5.308,Z -70.236,A -90.000,B 90.000,C 0.000} C_DIS
LIN {X -108.686,Y -5.308,Z -70.176,A -90.000,B 90.000,C 0.000} C_DIS
LIN {X -109.660,Y -5.308,Z -69.071,A -90.000,B 90.000,C 0.000} C_DIS
LIN {X -109.713,Y -5.308,Z -69.011,A -90.000,B 90.000,C 0.000} C_DIS
LIN {X -109.740,Y -5.308,Z -68.980,A -90.000,B 90.000,C 0.000} C_DIS
LIN {X -110.014,Y -5.308,Z -68.625,A -90.000,B 90.000,C 0.000} C_DIS
LIN {X -110.024,Y -5.308,Z -68.610,A -90.000,B 90.000,C 0.000} C_DIS
LIN {X -110.577,Y -5.308,Z -67.830,A -90.000,B 90.000,C 0.000} C_DIS
LIN {X -110.866,Y -5.308,Z -67.422,A -90.000,B 90.000,C 0.000} C_DIS
LIN {X -110.987,Y -5.308,Z -67.224,A -90.000,B 90.000,C 0.000} C_DIS
LIN {X -111.104,Y -5.308,Z -67.027,A -90.000,B 90.000,C 0.000} C_DIS
LIN {X -111.353,Y -5.308,Z -66.580,A -90.000,B 90.000,C 0.000} C_DIS
LIN {X -111.814,Y -5.308,Z -65.753,A -90.000,B 90.000,C 0.000} C_DIS
LIN {X -111.830,Y -5.308,Z -65.720,A -90.000,B 90.000,C 0.000} C_DIS
LIN {X -112.003,Y -5.308,Z -65.338,A -90.000,B 90.000,C 0.000} C_DIS
LIN {X -112.040,Y -5.308,Z -65.255,A -90.000,B 90.000,C 0.000} C_DIS
LIN {X -112.139,Y -5.308,Z -65.033,A -90.000,B 90.000,C 0.000} C_DIS
LIN {X -112.644,Y -5.308,Z -63.877,A -90.000,B 90.000,C 0.000} C_DIS
LIN {X -112.758,Y -5.308,Z -63.566,A -90.000,B 90.000,C 0.000} C_DIS
LIN {X -113.266,Y -5.308,Z -62.193,A -90.000,B 90.000,C 0.000} C_DIS
LIN {X -113.526,Y -5.308,Z -61.421,A -90.000,B 90.000,C 0.000} C_DIS
LIN {X -113.873,Y -5.308,Z -60.396,A -90.000,B 90.000,C 0.000} C_DIS
LIN {X -114.289,Y -5.308,Z -59.135,A -90.000,B 90.000,C 0.000} C_DIS
LIN {X -114.471,Y -5.308,Z -58.583,A -90.000,B 90.000,C 0.000} C_DIS
LIN {X -115.055,Y -5.308,Z -56.889,A -90.000,B 90.000,C 0.000} C_DIS
LIN {X -115.070,Y -5.308,Z -56.846,A -90.000,B 90.000,C 0.000} C_DIS
LIN {X -115.081,Y -5.308,Z -56.817,A -90.000,B 90.000,C 0.000} C_DIS
LIN {X -115.131,Y -5.308,Z -56.686,A -90.000,B 90.000,C 0.000} C_DIS
LIN {X -115.588,Y -5.308,Z -55.480,A -90.000,B 90.000,C 0.000} C_DIS
LIN {X -115.675,Y -5.308,Z -55.258,A -90.000,B 90.000,C 0.000} C_DIS
LIN {X -116.071,Y -5.308,Z -54.236,A -90.000,B 90.000,C 0.000} C_DIS
LIN {X -116.235,Y -5.308,Z -53.827,A -90.000,B 90.000,C 0.000} C_DIS
LIN {X -116.501,Y -5.308,Z -53.077,A -90.000,B 90.000,C 0.000} C_DIS
LIN {X -116.695,Y -5.308,Z -52.552,A -90.000,B 90.000,C 0.000} C_DIS
LIN {X -116.763,Y -5.308,Z -52.344,A -90.000,B 90.000,C 0.000} C_DIS
LIN {X -116.836,Y -5.308,Z -52.119,A -90.000,B 90.000,C 0.000} C_DIS
LIN {X -116.978,Y -5.308,Z -51.576,A -90.000,B 90.000,C 0.000} C_DIS
LIN {X -117.134,Y -5.308,Z -51.004,A -90.000,B 90.000,C 0.000} C_DIS
LIN {X -117.188,Y -5.308,Z -50.747,A -90.000,B 90.000,C 0.000} C_DIS
LIN {X -117.228,Y -5.308,Z -50.559,A -90.000,B 90.000,C 0.000} C_DIS
LIN {X -117.253,Y -5.308,Z -50.297,A -90.000,B 90.000,C 0.000} C_DIS
LIN {X -117.271,Y -5.308,Z -50.105,A -90.000,B 90.000,C 0.000} C_DIS
LIN {X -117.301,Y -5.308,Z -49.719,A -90.000,B 90.000,C 0.000} C_DIS
LIN {X -117.344,Y -5.308,Z -49.161,A -90.000,B 90.000,C 0.000} C_DIS
LIN {X -117.346,Y -5.308,Z -49.086,A -90.000,B 90.000,C 0.000} C_DIS
LIN {X -117.350,Y -5.308,Z -48.972,A -90.000,B 90.000,C 0.000} C_DIS
LIN {X -117.349,Y -5.308,Z -48.972,A -90.000,B 90.000,C 0.000} C_DIS
LIN {X -117.339,Y -5.308,Z -48.532,A -90.000,B 90.000,C 0.000} C_DIS
LIN {X -117.274,Y -5.308,Z -47.742,A -90.000,B 90.000,C 0.000} C_DIS
LIN {X -117.270,Y -5.308,Z -47.696,A -90.000,B 90.000,C 0.000} C_DIS
LIN {X -117.266,Y -5.308,Z -47.668,A -90.000,B 90.000,C 0.000} C_DIS
LIN {X -117.210,Y -5.308,Z -47.259,A -90.000,B 90.000,C 0.000} C_DIS
LIN {X -117.206,Y -5.308,Z -47.240,A -90.000,B 90.000,C 0.000} C_DIS
LIN {X -117.193,Y -5.308,Z -47.165,A -90.000,B 90.000,C 0.000} C_DIS
LIN {X -117.134,Y -5.308,Z -46.838,A -90.000,B 90.000,C 0.000} C_DIS
LIN {X -117.154,Y -5.308,Z -46.783,A -90.000,B 90.000,C 0.000} C_DIS
LIN {X -117.155,Y -5.308,Z -46.780,A -90.000,B 90.000,C 0.000} C_DIS
LIN {X -117.261,Y -5.308,Z -46.492,A -90.000,B 90.000,C 0.000} C_DIS
LIN {X -117.275,Y -5.308,Z -46.452,A -90.000,B 90.000,C 0.000} C_DIS
LIN {X -117.417,Y -5.308,Z -46.035,A -90.000,B 90.000,C 0.000} C_DIS
LIN {X -117.431,Y -5.308,Z -45.993,A -90.000,B 90.000,C 0.000} C_DIS
LIN {X -117.590,Y -5.308,Z -45.524,A -90.000,B 90.000,C 0.000} C_DIS
LIN {X -117.599,Y -5.308,Z -45.489,A -90.000,B 90.000,C 0.000} C_DIS
LIN {X -117.727,Y -5.308,Z -45.030,A -90.000,B 90.000,C 0.000} C_DIS
LIN {X -117.734,Y -5.308,Z -45.003,A -90.000,B 90.000,C 0.000} C_DIS
LIN {X -117.743,Y -5.308,Z -44.964,A -90.000,B 90.000,C 0.000} C_DIS
LIN {X -117.821,Y -5.308,Z -44.656,A -90.000,B 90.000,C 0.000} C_DIS
LIN {X -117.874,Y -5.308,Z -44.447,A -90.000,B 90.000,C 0.000} C_DIS
LIN {X -117.910,Y -5.308,Z -44.255,A -90.000,B 90.000,C 0.000} C_DIS
LIN {X -117.967,Y -5.308,Z -43.952,A -90.000,B 90.000,C 0.000} C_DIS
LIN {X -117.999,Y -5.308,Z -43.760,A -90.000,B 90.000,C 0.000} C_DIS
LIN {X -118.046,Y -5.308,Z -43.483,A -90.000,B 90.000,C 0.000} C_DIS
LIN {X -118.057,Y -5.308,Z -43.358,A -90.000,B 90.000,C 0.000} C_DIS
LIN {X -118.075,Y -5.308,Z -43.169,A -90.000,B 90.000,C 0.000} C_DIS
LIN {X -118.085,Y -5.308,Z -43.060,A -90.000,B 90.000,C 0.000} C_DIS
LIN {X -118.092,Y -5.308,Z -42.991,A -90.000,B 90.000,C 0.000} C_DIS
LIN {X -118.118,Y -5.308,Z -42.607,A -90.000,B 90.000,C 0.000} C_DIS
LIN {X -118.125,Y -5.308,Z -42.500,A -90.000,B 90.000,C 0.000} C_DIS
LIN {X -118.131,Y -5.308,Z -42.130,A -90.000,B 90.000,C 0.000} C_DIS
LIN {X -118.132,Y -5.308,Z -42.033,A -90.000,B 90.000,C 0.000} C_DIS
LIN {X -118.113,Y -5.308,Z -41.654,A -90.000,B 90.000,C 0.000} C_DIS
LIN {X -118.109,Y -5.308,Z -41.572,A -90.000,B 90.000,C 0.000} C_DIS
LIN {X -118.092,Y -5.308,Z -41.377,A -90.000,B 90.000,C 0.000} C_DIS
LIN {X -118.076,Y -5.308,Z -41.197,A -90.000,B 90.000,C 0.000} C_DIS
LIN {X -118.071,Y -5.308,Z -41.145,A -90.000,B 90.000,C 0.000} C_DIS
LIN {X -118.067,Y -5.308,Z -41.107,A -90.000,B 90.000,C 0.000} C_DIS
LIN {X -118.043,Y -5.308,Z -40.919,A -90.000,B 90.000,C 0.000} C_DIS
LIN {X -118.020,Y -5.308,Z -40.745,A -90.000,B 90.000,C 0.000} C_DIS
LIN {X -118.003,Y -5.308,Z -40.644,A -90.000,B 90.000,C 0.000} C_DIS
LIN {X -117.948,Y -5.308,Z -40.318,A -90.000,B 90.000,C 0.000} C_DIS
LIN {X -117.920,Y -5.308,Z -40.200,A -90.000,B 90.000,C 0.000} C_DIS
LIN {X -117.843,Y -5.308,Z -39.875,A -90.000,B 90.000,C 0.000} C_DIS
LIN {X -117.813,Y -5.308,Z -39.775,A -90.000,B 90.000,C 0.000} C_DIS
LIN {X -117.728,Y -5.308,Z -39.499,A -90.000,B 90.000,C 0.000} C_DIS
LIN {X -117.683,Y -5.308,Z -39.375,A -90.000,B 90.000,C 0.000} C_DIS
LIN {X -117.575,Y -5.308,Z -39.070,A -90.000,B 90.000,C 0.000} C_DIS
LIN {X -117.556,Y -5.308,Z -39.026,A -90.000,B 90.000,C 0.000} C_DIS
LIN {X -117.523,Y -5.308,Z -38.947,A -90.000,B 90.000,C 0.000} C_DIS
LIN {X -117.427,Y -5.308,Z -38.748,A -90.000,B 90.000,C 0.000} C_DIS
LIN {X -117.400,Y -5.308,Z -38.694,A -90.000,B 90.000,C 0.000} C_DIS
LIN {X -117.444,Y -5.308,Z -38.581,A -90.000,B 90.000,C 0.000} C_DIS
LIN {X -117.489,Y -5.308,Z -38.464,A -90.000,B 90.000,C 0.000} C_DIS
LIN {X -117.521,Y -5.308,Z -38.369,A -90.000,B 90.000,C 0.000} C_DIS
LIN {X -117.622,Y -5.308,Z -38.070,A -90.000,B 90.000,C 0.000} C_DIS
LIN {X -117.717,Y -5.308,Z -37.761,A -90.000,B 90.000,C 0.000} C_DIS
LIN {X -117.766,Y -5.308,Z -37.605,A -90.000,B 90.000,C 0.000} C_DIS
LIN {X -117.789,Y -5.308,Z -37.520,A -90.000,B 90.000,C 0.000} C_DIS
LIN {X -117.820,Y -5.308,Z -37.404,A -90.000,B 90.000,C 0.000} C_DIS
LIN {X -117.896,Y -5.308,Z -37.116,A -90.000,B 90.000,C 0.000} C_DIS
LIN {X -117.908,Y -5.308,Z -37.071,A -90.000,B 90.000,C 0.000} C_DIS
LIN {X -118.012,Y -5.308,Z -36.614,A -90.000,B 90.000,C 0.000} C_DIS
LIN {X -118.015,Y -5.308,Z -36.601,A -90.000,B 90.000,C 0.000} C_DIS
LIN {X -118.016,Y -5.308,Z -36.598,A -90.000,B 90.000,C 0.000} C_DIS
LIN {X -118.016,Y -5.308,Z -36.596,A -90.000,B 90.000,C 0.000} C_DIS
LIN {X -118.058,Y -5.308,Z -36.331,A -90.000,B 90.000,C 0.000} C_DIS
LIN {X -118.063,Y -5.308,Z -36.301,A -90.000,B 90.000,C 0.000} C_DIS
LIN {X -118.114,Y -5.308,Z -35.874,A -90.000,B 90.000,C 0.000} C_DIS
LIN {X -118.121,Y -5.308,Z -35.822,A -90.000,B 90.000,C 0.000} C_DIS
LIN {X -118.136,Y -5.308,Z -35.595,A -90.000,B 90.000,C 0.000} C_DIS
LIN {X -118.139,Y -5.308,Z -35.543,A -90.000,B 90.000,C 0.000} C_DIS
LIN {X -118.146,Y -5.308,Z -35.156,A -90.000,B 90.000,C 0.000} C_DIS
LIN {X -118.147,Y -5.308,Z -35.061,A -90.000,B 90.000,C 0.000} C_DIS
LIN {X -118.147,Y -5.308,Z -35.022,A -90.000,B 90.000,C 0.000} C_DIS
LIN {X -118.147,Y -5.308,Z -34.988,A -90.000,B 90.000,C 0.000} C_DIS
LIN {X -118.146,Y -5.308,Z -34.915,A -90.000,B 90.000,C 0.000} C_DIS
LIN {X -118.146,Y -5.308,Z -34.883,A -90.000,B 90.000,C 0.000} C_DIS
LIN {X -118.145,Y -5.308,Z -34.852,A -90.000,B 90.000,C 0.000} C_DIS
LIN {X -118.144,Y -5.308,Z -34.778,A -90.000,B 90.000,C 0.000} C_DIS
LIN {X -118.143,Y -5.308,Z -34.742,A -90.000,B 90.000,C 0.000} C_DIS
LIN {X -118.142,Y -5.308,Z -34.703,A -90.000,B 90.000,C 0.000} C_DIS
LIN {X -118.138,Y -5.308,Z -34.606,A -90.000,B 90.000,C 0.000} C_DIS
LIN {X -118.121,Y -5.308,Z -34.227,A -90.000,B 90.000,C 0.000} C_DIS
LIN {X -118.116,Y -5.308,Z -34.174,A -90.000,B 90.000,C 0.000} C_DIS
LIN {X -118.094,Y -5.308,Z -33.943,A -90.000,B 90.000,C 0.000} C_DIS
LIN {X -118.089,Y -5.308,Z -33.907,A -90.000,B 90.000,C 0.000} C_DIS
LIN {X -118.080,Y -5.308,Z -33.848,A -90.000,B 90.000,C 0.000} C_DIS
LIN {X -118.018,Y -5.308,Z -33.436,A -90.000,B 90.000,C 0.000} C_DIS
